LIN {X 0,Y 374.396,Z 363.23,A -85,B 0,C 180,E1 -12882.407,E2 -12882.407} C_VEL
LIN {X 0,Y 374.739,Z 351.061,A -85,B 0,C 180,E1 -12882.778,E2 -12882.778} C_VEL
LIN {X 0,Y 374.257,Z 345.258,A -85,B 0,C 180,E1 -12882.93,E2 -12882.93} C_VEL
LIN {X 0,Y 369.029,Z 326.535,A -85,B 0,C 180,E1 -12883.548,E2 -12883.548} C_VEL
LIN {X 0,Y 368.498,Z 320.718,A -85,B 0,C 180,E1 -12883.688,E2 -12883.688} C_VEL
LIN {X 0,Y 369.139,Z 272.21,A -85,B 0,C 180,E1 -12884.631,E2 -12884.631} C_VEL
LIN {X 0,Y 364.648,Z 248.183,A -85,B 0,C 180,E1 -12885.359,E2 -12885.359} C_VEL
LIN {X 0,Y 364.36,Z 246.734,A -85,B 0,C 180,E1 -12885.446,E2 -12885.446} C_VEL
LIN {X 0,Y 361.947,Z 234.402,A -85,B 0,C 180,E1 -12888.759,E2 -12888.759} C_VEL
LIN {X 0,Y 361.881,Z 234.409,A -85,B 0,C 180,E1 -12892.856,E2 -12892.856} C_VEL
LIN {X 0,Y 361.903,Z 234.406,A -85,B 0,C 180,E1 -12896.529,E2 -12896.529} C_VEL
LIN {X 0,Y 361.869,Z 234.408,A -85,B 0,C 180,E1 -12900.328,E2 -12900.328} C_VEL
LIN {X 0,Y 361.856,Z 234.409,A -85,B 0,C 180,E1 -12904.28,E2 -12904.28} C_VEL
LIN {X 0,Y 361.865,Z 234.407,A -85,B 0,C 180,E1 -12907.223,E2 -12907.223} C_VEL
LIN {X 0,Y 361.837,Z 234.415,A -85,B 0,C 180,E1 -12910.755,E2 -12910.755} C_VEL
LIN {X 0,Y 361.847,Z 234.411,A -85,B 0,C 180,E1 -12914.364,E2 -12914.364} C_VEL
LIN {X 0,Y 361.836,Z 234.409,A -85,B 0,C 180,E1 -12917.568,E2 -12917.568} C_VEL
LIN {X 0,Y 361.867,Z 234.409,A -85,B 0,C 180,E1 -12920.974,E2 -12920.974} C_VEL
LIN {X 0,Y 361.875,Z 234.411,A -85,B 0,C 180,E1 -12924.655,E2 -12924.655} C_VEL
LIN {X 0,Y 361.839,Z 234.413,A -85,B 0,C 180,E1 -12928.37,E2 -12928.37} C_VEL
LIN {X 0,Y 361.909,Z 234.403,A -85,B 0,C 180,E1 -12932.221,E2 -12932.221} C_VEL
LIN {X 0,Y 361.928,Z 234.404,A -85,B 0,C 180,E1 -12934.71,E2 -12934.71} C_VEL
LIN {X 0,Y 361.894,Z 234.406,A -85,B 0,C 180,E1 -12938.347,E2 -12938.347} C_VEL
LIN {X 0,Y 361.968,Z 234.394,A -85,B 0,C 180,E1 -12942.061,E2 -12942.061} C_VEL
LIN {X 0,Y 361.999,Z 234.391,A -85,B 0,C 180,E1 -12946.101,E2 -12946.101} C_VEL
LIN {X 0,Y 362.001,Z 234.39,A -85,B 0,C 180,E1 -12949.937,E2 -12949.937} C_VEL
LIN {X 0,Y 362.136,Z 234.373,A -85,B 0,C 180,E1 -12953.313,E2 -12953.313} C_VEL
LIN {X 0,Y 362.281,Z 234.354,A -85,B 0,C 180,E1 -12957.776,E2 -12957.776} C_VEL
LIN {X 0,Y 362.425,Z 234.337,A -85,B 0,C 180,E1 -12960,E2 -12960} C_VEL
LIN {X 0,Y 362.278,Z 234.357,A -85,B 0,C 180,E1 -12962.223,E2 -12962.223} C_VEL
LIN {X 0,Y 362.173,Z 234.373,A -85,B 0,C 180,E1 -12966.686,E2 -12966.686} C_VEL
LIN {X 0,Y 362.075,Z 234.383,A -85,B 0,C 180,E1 -12968.933,E2 -12968.933} C_VEL
LIN {X 0,Y 361.96,Z 234.398,A -85,B 0,C 180,E1 -12972.332,E2 -12972.332} C_VEL
LIN {X 0,Y 361.962,Z 234.4,A -85,B 0,C 180,E1 -12974.62,E2 -12974.62} C_VEL
LIN {X 0,Y 361.911,Z 234.402,A -85,B 0,C 180,E1 -12978.102,E2 -12978.102} C_VEL
LIN {X 0,Y 361.861,Z 234.406,A -85,B 0,C 180,E1 -12981.655,E2 -12981.655} C_VEL
LIN {X 0,Y 361.894,Z 234.403,A -85,B 0,C 180,E1 -12985.293,E2 -12985.293} C_VEL
LIN {X 0,Y 361.855,Z 234.409,A -85,B 0,C 180,E1 -12989.074,E2 -12989.074} C_VEL
LIN {X 0,Y 361.849,Z 234.41,A -85,B 0,C 180,E1 -12992.945,E2 -12992.945} C_VEL
LIN {X 0,Y 361.868,Z 234.405,A -85,B 0,C 180,E1 -12995.637,E2 -12995.637} C_VEL
LIN {X 0,Y 361.826,Z 234.413,A -85,B 0,C 180,E1 -12999.018,E2 -12999.018} C_VEL
LIN {X 0,Y 361.833,Z 234.413,A -85,B 0,C 180,E1 -13002.829,E2 -13002.829} C_VEL
LIN {X 0,Y 361.818,Z 234.413,A -85,B 0,C 180,E1 -13005.947,E2 -13005.947} C_VEL
LIN {X 0,Y 361.83,Z 234.411,A -85,B 0,C 180,E1 -13009.246,E2 -13009.246} C_VEL
LIN {X 0,Y 361.87,Z 234.409,A -85,B 0,C 180,E1 -13012.776,E2 -13012.776} C_VEL
LIN {X 0,Y 361.855,Z 234.407,A -85,B 0,C 180,E1 -13015.72,E2 -13015.72} C_VEL
LIN {X 0,Y 361.874,Z 234.409,A -85,B 0,C 180,E1 -13019.672,E2 -13019.672} C_VEL
LIN {X 0,Y 361.925,Z 234.53,A -85,B 0,C 180,E1 -13021.156,E2 -13021.156} C_VEL
LIN {X 0,Y 363.889,Z 244.234,A -85,B 0,C 180,E1 -13023.627,E2 -13023.627} C_VEL
LIN {X 0,Y 365.118,Z 252.079,A -85,B 0,C 180,E1 -13025.553,E2 -13025.553} C_VEL
LIN {X 0,Y 364.017,Z 265.513,A -85,B 0,C 180,E1 -13028.609,E2 -13028.609} C_VEL
LIN {X 0,Y 368.872,Z 299.067,A -85,B 0,C 180,E1 -13029.543,E2 -13029.543} C_VEL
LIN {X 0,Y 367.713,Z 373.609,A -85,B 0,C 180,E1 -13031.005,E2 -13031.005} C_VEL
LIN {X 0,Y 367.121,Z 386.917,A -85,B 0,C 180,E1 -13031.478,E2 -13031.478} C_VEL
LIN {X 0,Y 366.35,Z 399.141,A -85,B 0,C 180,E1 -13032.125,E2 -13032.125} C_VEL
LIN {X 0,Y 365.487,Z 410.647,A -85,B 0,C 180,E1 -13032.948,E2 -13032.948} C_VEL
LIN {X 0,Y 364.414,Z 422.442,A -85,B 0,C 180,E1 -13034.049,E2 -13034.049} C_VEL
LIN {X 0,Y 363.531,Z 432.403,A -85,B 0,C 180,E1 -13035.218,E2 -13035.218} C_VEL
LIN {X 0,Y 362.727,Z 441.68,A -85,B 0,C 180,E1 -13036.555,E2 -13036.555} C_VEL
LIN {X 0,Y 361.986,Z 449.644,A -85,B 0,C 180,E1 -13037.953,E2 -13037.953} C_VEL
LIN {X 0,Y 361.295,Z 457.417,A -85,B 0,C 180,E1 -13039.634,E2 -13039.634} C_VEL
LIN {X 0,Y 360.779,Z 464.561,A -85,B 0,C 180,E1 -13041.599,E2 -13041.599} C_VEL
LIN {X 0,Y 360.498,Z 469.31,A -85,B 0,C 180,E1 -13043.283,E2 -13043.283} C_VEL
LIN {X 0,Y 360.35,Z 472.934,A -85,B 0,C 180,E1 -13044.965,E2 -13044.965} C_VEL
LIN {X 0,Y 360.301,Z 475.537,A -85,B 0,C 180,E1 -13046.645,E2 -13046.645} C_VEL
LIN {X 0,Y 360.266,Z 476.761,A -85,B 0,C 180,E1 -13047.764,E2 -13047.764} C_VEL
LIN {X 0,Y 360.317,Z 477.556,A -85,B 0,C 180,E1 -13048.882,E2 -13048.882} C_VEL
LIN {X 0,Y 360.359,Z 477.936,A -85,B 0,C 180,E1 -13050,E2 -13050} C_VEL
LIN {X 0,Y 360.303,Z 477.928,A -85,B 0,C 180,E1 -13051.118,E2 -13051.118} C_VEL
LIN {X 0,Y 360.262,Z 477.537,A -85,B 0,C 180,E1 -13052.236,E2 -13052.236} C_VEL
LIN {X 0,Y 360.296,Z 476.738,A -85,B 0,C 180,E1 -13053.355,E2 -13053.355} C_VEL
LIN {X 0,Y 360.348,Z 475.51,A -85,B 0,C 180,E1 -13054.474,E2 -13054.474} C_VEL
LIN {X 0,Y 360.432,Z 473.128,A -85,B 0,C 180,E1 -13056.043,E2 -13056.043} C_VEL
LIN {X 0,Y 360.699,Z 469.313,A -85,B 0,C 180,E1 -13057.839,E2 -13057.839} C_VEL
LIN {X 0,Y 361.175,Z 464.617,A -85,B 0,C 180,E1 -13059.52,E2 -13059.52} C_VEL
LIN {X 0,Y 361.972,Z 457.568,A -85,B 0,C 180,E1 -13061.479,E2 -13061.479} C_VEL
LIN {X 0,Y 362.996,Z 449.946,A -85,B 0,C 180,E1 -13063.15,E2 -13063.15} C_VEL
LIN {X 0,Y 364.15,Z 440.878,A -85,B 0,C 180,E1 -13064.737,E2 -13064.737} C_VEL
LIN {X 0,Y 365.288,Z 430.537,A -85,B 0,C 180,E1 -13066.199,E2 -13066.199} C_VEL
LIN {X 0,Y 366.645,Z 419.502,A -85,B 0,C 180,E1 -13067.428,E2 -13067.428} C_VEL
LIN {X 0,Y 367.739,Z 408.708,A -85,B 0,C 180,E1 -13068.381,E2 -13068.381} C_VEL
LIN {X 0,Y 368.907,Z 396.811,A -85,B 0,C 180,E1 -13069.186,E2 -13069.186} C_VEL
LIN {X 0,Y 369.813,Z 383.937,A -85,B 0,C 180,E1 -13069.822,E2 -13069.822} C_VEL
LIN {X 0,Y 370.412,Z 370.747,A -85,B 0,C 180,E1 -13070.235,E2 -13070.235} C_VEL
LIN {X 0,Y 371.679,Z 298.745,A -85,B 0,C 180,E1 -13071.649,E2 -13071.649} C_VEL
LIN {X 0,Y 366.907,Z 272.712,A -85,B 0,C 180,E1 -13072.526,E2 -13072.526} C_VEL
LIN {X 0,Y 365.363,Z 265.186,A -85,B 0,C 180,E1 -13072.806,E2 -13072.806} C_VEL
LIN {X 0,Y 366.337,Z 255.911,A -85,B 0,C 180,E1 -13074.965,E2 -13074.965} C_VEL
LIN {X 0,Y 364.479,Z 245.888,A -85,B 0,C 180,E1 -13077.566,E2 -13077.566} C_VEL
LIN {X 0,Y 362.218,Z 235.875,A -85,B 0,C 180,E1 -13080.296,E2 -13080.296} C_VEL
LIN {X 0,Y 361.896,Z 234.407,A -85,B 0,C 180,E1 -13080.708,E2 -13080.708} C_VEL
LIN {X 0,Y 361.855,Z 234.41,A -85,B 0,C 180,E1 -13084.28,E2 -13084.28} C_VEL
LIN {X 0,Y 361.864,Z 234.411,A -85,B 0,C 180,E1 -13087.223,E2 -13087.223} C_VEL
LIN {X 0,Y 361.835,Z 234.413,A -85,B 0,C 180,E1 -13090.755,E2 -13090.755} C_VEL
LIN {X 0,Y 361.817,Z 234.414,A -85,B 0,C 180,E1 -13094.369,E2 -13094.369} C_VEL
LIN {X 0,Y 361.831,Z 234.415,A -85,B 0,C 180,E1 -13097.569,E2 -13097.569} C_VEL
LIN {X 0,Y 361.844,Z 234.413,A -85,B 0,C 180,E1 -13101.572,E2 -13101.572} C_VEL
LIN {X 0,Y 361.874,Z 234.405,A -85,B 0,C 180,E1 -13104.655,E2 -13104.655} C_VEL
LIN {X 0,Y 361.838,Z 234.41,A -85,B 0,C 180,E1 -13108.371,E2 -13108.371} C_VEL
LIN {X 0,Y 361.866,Z 234.401,A -85,B 0,C 180,E1 -13110.952,E2 -13110.952} C_VEL
LIN {X 0,Y 361.902,Z 234.396,A -85,B 0,C 180,E1 -13114.708,E2 -13114.708} C_VEL
LIN {X 0,Y 361.862,Z 234.403,A -85,B 0,C 180,E1 -13118.345,E2 -13118.345} C_VEL
LIN {X 0,Y 361.921,Z 234.398,A -85,B 0,C 180,E1 -13122.085,E2 -13122.085} C_VEL
LIN {X 0,Y 361.963,Z 234.398,A -85,B 0,C 180,E1 -13125.38,E2 -13125.38} C_VEL
LIN {X 0,Y 361.971,Z 234.388,A -85,B 0,C 180,E1 -13128.804,E2 -13128.804} C_VEL
LIN {X 0,Y 362.125,Z 234.369,A -85,B 0,C 180,E1 -13132.192,E2 -13132.192} C_VEL
LIN {X 0,Y 362.115,Z 234.373,A -85,B 0,C 180,E1 -13134.431,E2 -13134.431} C_VEL
LIN {X 0,Y 362.272,Z 234.35,A -85,B 0,C 180,E1 -13137.776,E2 -13137.776} C_VEL
LIN {X 0,Y 362.425,Z 234.338,A -85,B 0,C 180,E1 -13140,E2 -13140} C_VEL
LIN {X 0,Y 362.279,Z 234.35,A -85,B 0,C 180,E1 -13142.224,E2 -13142.224} C_VEL
LIN {X 0,Y 362.137,Z 234.373,A -85,B 0,C 180,E1 -13146.687,E2 -13146.687} C_VEL
LIN {X 0,Y 362.001,Z 234.391,A -85,B 0,C 180,E1 -13150.063,E2 -13150.063} C_VEL
LIN {X 0,Y 361.999,Z 234.388,A -85,B 0,C 180,E1 -13153.899,E2 -13153.899} C_VEL
LIN {X 0,Y 361.929,Z 234.399,A -85,B 0,C 180,E1 -13156.934,E2 -13156.934} C_VEL
LIN {X 0,Y 361.895,Z 234.402,A -85,B 0,C 180,E1 -13160.461,E2 -13160.461} C_VEL
LIN {X 0,Y 361.895,Z 234.403,A -85,B 0,C 180,E1 -13164.113,E2 -13164.113} C_VEL
LIN {X 0,Y 361.942,Z 234.391,A -85,B 0,C 180,E1 -13166.721,E2 -13166.721} C_VEL
LIN {X 0,Y 361.874,Z 234.402,A -85,B 0,C 180,E1 -13170.328,E2 -13170.328} C_VEL
LIN {X 0,Y 361.856,Z 234.408,A -85,B 0,C 180,E1 -13174.281,E2 -13174.281} C_VEL
LIN {X 0,Y 361.871,Z 234.408,A -85,B 0,C 180,E1 -13177.224,E2 -13177.224} C_VEL
LIN {X 0,Y 361.836,Z 234.412,A -85,B 0,C 180,E1 -13180.755,E2 -13180.755} C_VEL
LIN {X 0,Y 361.821,Z 234.415,A -85,B 0,C 180,E1 -13184.368,E2 -13184.368} C_VEL
LIN {X 0,Y 361.833,Z 234.412,A -85,B 0,C 180,E1 -13187.569,E2 -13187.569} C_VEL
LIN {X 0,Y 361.846,Z 234.42,A -85,B 0,C 180,E1 -13191.572,E2 -13191.572} C_VEL
LIN {X 0,Y 361.876,Z 234.412,A -85,B 0,C 180,E1 -13194.655,E2 -13194.655} C_VEL
LIN {X 0,Y 361.89,Z 234.581,A -85,B 0,C 180,E1 -13197.638,E2 -13197.638} C_VEL
LIN {X 0,Y 364.482,Z 246.196,A -85,B 0,C 180,E1 -13200.943,E2 -13200.943} C_VEL
LIN {X 0,Y 364.656,Z 247.154,A -85,B 0,C 180,E1 -13201.195,E2 -13201.195} C_VEL
LIN {X 0,Y 368.325,Z 257.097,A -85,B 0,C 180,E1 -13201.675,E2 -13201.675} C_VEL
LIN {X 0,Y 372.157,Z 273.927,A -85,B 0,C 180,E1 -13202.297,E2 -13202.297} C_VEL
LIN {X 0,Y 370.619,Z 354.332,A -85,B 0,C 180,E1 -13203.881,E2 -13203.881} C_VEL
LIN {X 0,Y 369.973,Z 367.682,A -85,B 0,C 180,E1 -13204.358,E2 -13204.358} C_VEL
LIN {X 0,Y 369.232,Z 379.987,A -85,B 0,C 180,E1 -13205.019,E2 -13205.019} C_VEL
LIN {X 0,Y 368.134,Z 392.32,A -85,B 0,C 180,E1 -13205.916,E2 -13205.916} C_VEL
LIN {X 0,Y 367.068,Z 403.069,A -85,B 0,C 180,E1 -13206.937,E2 -13206.937} C_VEL
LIN {X 0,Y 365.742,Z 413.323,A -85,B 0,C 180,E1 -13208.142,E2 -13208.142} C_VEL
LIN {X 0,Y 364.786,Z 422.027,A -85,B 0,C 180,E1 -13209.414,E2 -13209.414} C_VEL
LIN {X 0,Y 363.735,Z 430.01,A -85,B 0,C 180,E1 -13210.824,E2 -13210.824} C_VEL
LIN {X 0,Y 362.722,Z 437.778,A -85,B 0,C 180,E1 -13212.523,E2 -13212.523} C_VEL
LIN {X 0,Y 361.904,Z 443.979,A -85,B 0,C 180,E1 -13214.224,E2 -13214.224} C_VEL
LIN {X 0,Y 361.308,Z 448.882,A -85,B 0,C 180,E1 -13215.928,E2 -13215.928} C_VEL
LIN {X 0,Y 360.865,Z 452.641,A -85,B 0,C 180,E1 -13217.63,E2 -13217.63} C_VEL
LIN {X 0,Y 360.603,Z 454.574,A -85,B 0,C 180,E1 -13218.761,E2 -13218.761} C_VEL
LIN {X 0,Y 360.406,Z 456.08,A -85,B 0,C 180,E1 -13219.892,E2 -13219.892} C_VEL
LIN {X 0,Y 360.346,Z 457.127,A -85,B 0,C 180,E1 -13221.024,E2 -13221.024} C_VEL
LIN {X 0,Y 360.356,Z 458.051,A -85,B 0,C 180,E1 -13223.28,E2 -13223.28} C_VEL
LIN {X 0,Y 360.339,Z 457.93,A -85,B 0,C 180,E1 -13224.404,E2 -13224.404} C_VEL
LIN {X 0,Y 360.337,Z 457.379,A -85,B 0,C 180,E1 -13225.525,E2 -13225.525} C_VEL
LIN {X 0,Y 360.368,Z 455.116,A -85,B 0,C 180,E1 -13227.765,E2 -13227.765} C_VEL
LIN {X 0,Y 360.561,Z 452.313,A -85,B 0,C 180,E1 -13229.442,E2 -13229.442} C_VEL
LIN {X 0,Y 360.77,Z 448.504,A -85,B 0,C 180,E1 -13231.116,E2 -13231.116} C_VEL
LIN {X 0,Y 361.196,Z 443.574,A -85,B 0,C 180,E1 -13232.788,E2 -13232.788} C_VEL
LIN {X 0,Y 361.732,Z 437.388,A -85,B 0,C 180,E1 -13234.457,E2 -13234.457} C_VEL
LIN {X 0,Y 362.497,Z 429.658,A -85,B 0,C 180,E1 -13236.121,E2 -13236.121} C_VEL
LIN {X 0,Y 363.56,Z 419.993,A -85,B 0,C 180,E1 -13237.777,E2 -13237.777} C_VEL
LIN {X 0,Y 364.5,Z 410.002,A -85,B 0,C 180,E1 -13239.153,E2 -13239.153} C_VEL
LIN {X 0,Y 365.488,Z 398.682,A -85,B 0,C 180,E1 -13240.386,E2 -13240.386} C_VEL
LIN {X 0,Y 366.334,Z 387.589,A -85,B 0,C 180,E1 -13241.341,E2 -13241.341} C_VEL
LIN {X 0,Y 367.092,Z 375.196,A -85,B 0,C 180,E1 -13242.157,E2 -13242.157} C_VEL
LIN {X 0,Y 367.633,Z 362.16,A -85,B 0,C 180,E1 -13242.762,E2 -13242.762} C_VEL
LIN {X 0,Y 367.993,Z 349.854,A -85,B 0,C 180,E1 -13243.124,E2 -13243.124} C_VEL
LIN {X 0,Y 368.498,Z 320.718,A -85,B 0,C 180,E1 -13243.688,E2 -13243.688} C_VEL
LIN {X 0,Y 367.969,Z 314.906,A -85,B 0,C 180,E1 -13243.831,E2 -13243.831} C_VEL
LIN {X 0,Y 362.777,Z 296.203,A -85,B 0,C 180,E1 -13244.477,E2 -13244.477} C_VEL
LIN {X 0,Y 362.288,Z 290.391,A -85,B 0,C 180,E1 -13244.621,E2 -13244.621} C_VEL
LIN {X 0,Y 362.466,Z 273.403,A -85,B 0,C 180,E1 -13244.961,E2 -13244.961} C_VEL
LIN {X 0,Y 358.093,Z 249.854,A -85,B 0,C 180,E1 -13245.691,E2 -13245.691} C_VEL
LIN {X 0,Y 357.227,Z 246.955,A -85,B 0,C 180,E1 -13245.837,E2 -13245.837} C_VEL
LIN {X 0,Y 354.899,Z 235.278,A -85,B 0,C 180,E1 -13249.071,E2 -13249.071} C_VEL
LIN {X 0,Y 354.818,Z 235.285,A -85,B 0,C 180,E1 -13252.107,E2 -13252.107} C_VEL
LIN {X 0,Y 354.866,Z 235.278,A -85,B 0,C 180,E1 -13255.83,E2 -13255.83} C_VEL
LIN {X 0,Y 354.809,Z 235.285,A -85,B 0,C 180,E1 -13259.683,E2 -13259.683} C_VEL
LIN {X 0,Y 354.816,Z 235.284,A -85,B 0,C 180,E1 -13263.684,E2 -13263.684} C_VEL
LIN {X 0,Y 354.8,Z 235.29,A -85,B 0,C 180,E1 -13266.459,E2 -13266.459} C_VEL
LIN {X 0,Y 354.826,Z 235.283,A -85,B 0,C 180,E1 -13269.423,E2 -13269.423} C_VEL
LIN {X 0,Y 354.79,Z 235.291,A -85,B 0,C 180,E1 -13272.867,E2 -13272.867} C_VEL
LIN {X 0,Y 354.769,Z 235.291,A -85,B 0,C 180,E1 -13276.104,E2 -13276.104} C_VEL
LIN {X 0,Y 354.786,Z 235.289,A -85,B 0,C 180,E1 -13279.178,E2 -13279.178} C_VEL
LIN {X 0,Y 354.807,Z 235.289,A -85,B 0,C 180,E1 -13282.402,E2 -13282.402} C_VEL
LIN {X 0,Y 354.813,Z 235.288,A -85,B 0,C 180,E1 -13284.941,E2 -13284.941} C_VEL
LIN {X 0,Y 354.794,Z 235.29,A -85,B 0,C 180,E1 -13288.405,E2 -13288.405} C_VEL
LIN {X 0,Y 354.847,Z 235.28,A -85,B 0,C 180,E1 -13291.618,E2 -13291.618} C_VEL
LIN {X 0,Y 354.899,Z 235.275,A -85,B 0,C 180,E1 -13294.172,E2 -13294.172} C_VEL
LIN {X 0,Y 354.837,Z 235.282,A -85,B 0,C 180,E1 -13297.894,E2 -13297.894} C_VEL
LIN {X 0,Y 354.923,Z 235.271,A -85,B 0,C 180,E1 -13301.891,E2 -13301.891} C_VEL
LIN {X 0,Y 354.943,Z 235.269,A -85,B 0,C 180,E1 -13305.981,E2 -13305.981} C_VEL
LIN {X 0,Y 354.957,Z 235.266,A -85,B 0,C 180,E1 -13309.735,E2 -13309.735} C_VEL
LIN {X 0,Y 355.099,Z 235.25,A -85,B 0,C 180,E1 -13313.18,E2 -13313.18} C_VEL
LIN {X 0,Y 355.244,Z 235.231,A -85,B 0,C 180,E1 -13317.732,E2 -13317.732} C_VEL
LIN {X 0,Y 355.374,Z 235.215,A -85,B 0,C 180,E1 -13320,E2 -13320} C_VEL
LIN {X 0,Y 355.241,Z 235.234,A -85,B 0,C 180,E1 -13322.268,E2 -13322.268} C_VEL
LIN {X 0,Y 355.139,Z 235.248,A -85,B 0,C 180,E1 -13326.819,E2 -13326.819} C_VEL
LIN {X 0,Y 355.016,Z 235.261,A -85,B 0,C 180,E1 -13329.112,E2 -13329.112} C_VEL
LIN {X 0,Y 354.922,Z 235.277,A -85,B 0,C 180,E1 -13332.581,E2 -13332.581} C_VEL
LIN {X 0,Y 354.888,Z 235.277,A -85,B 0,C 180,E1 -13336.096,E2 -13336.096} C_VEL
LIN {X 0,Y 354.844,Z 235.28,A -85,B 0,C 180,E1 -13339.676,E2 -13339.676} C_VEL
LIN {X 0,Y 354.825,Z 235.283,A -85,B 0,C 180,E1 -13343.337,E2 -13343.337} C_VEL
LIN {X 0,Y 354.814,Z 235.287,A -85,B 0,C 180,E1 -13346.958,E2 -13346.958} C_VEL
LIN {X 0,Y 354.799,Z 235.286,A -85,B 0,C 180,E1 -13349.684,E2 -13349.684} C_VEL
LIN {X 0,Y 354.787,Z 235.291,A -85,B 0,C 180,E1 -13352.333,E2 -13352.333} C_VEL
LIN {X 0,Y 354.822,Z 235.283,A -85,B 0,C 180,E1 -13355.699,E2 -13355.699} C_VEL
LIN {X 0,Y 354.768,Z 235.29,A -85,B 0,C 180,E1 -13359.413,E2 -13359.413} C_VEL
LIN {X 0,Y 354.786,Z 235.291,A -85,B 0,C 180,E1 -13362.867,E2 -13362.867} C_VEL
LIN {X 0,Y 354.767,Z 235.292,A -85,B 0,C 180,E1 -13366.104,E2 -13366.104} C_VEL
LIN {X 0,Y 354.782,Z 235.289,A -85,B 0,C 180,E1 -13369.178,E2 -13369.178} C_VEL
LIN {X 0,Y 354.811,Z 235.29,A -85,B 0,C 180,E1 -13372.402,E2 -13372.402} C_VEL
LIN {X 0,Y 354.812,Z 235.287,A -85,B 0,C 180,E1 -13374.941,E2 -13374.941} C_VEL
LIN {X 0,Y 354.794,Z 235.292,A -85,B 0,C 180,E1 -13378.405,E2 -13378.405} C_VEL
LIN {X 0,Y 354.879,Z 235.478,A -85,B 0,C 180,E1 -13380.875,E2 -13380.875} C_VEL
LIN {X 0,Y 356.852,Z 245.099,A -85,B 0,C 180,E1 -13383.382,E2 -13383.382} C_VEL
LIN {X 0,Y 358.18,Z 253.083,A -85,B 0,C 180,E1 -13385.389,E2 -13385.389} C_VEL
LIN {X 0,Y 357.143,Z 265.309,A -85,B 0,C 180,E1 -13388.226,E2 -13388.226} C_VEL
LIN {X 0,Y 362.12,Z 299.306,A -85,B 0,C 180,E1 -13389.2,E2 -13389.2} C_VEL
LIN {X 0,Y 360.906,Z 374.206,A -85,B 0,C 180,E1 -13390.705,E2 -13390.705} C_VEL
LIN {X 0,Y 360.227,Z 388.055,A -85,B 0,C 180,E1 -13391.221,E2 -13391.221} C_VEL
LIN {X 0,Y 359.396,Z 400.464,A -85,B 0,C 180,E1 -13391.915,E2 -13391.915} C_VEL
LIN {X 0,Y 358.382,Z 413.153,A -85,B 0,C 180,E1 -13392.893,E2 -13392.893} C_VEL
LIN {X 0,Y 357.306,Z 424.442,A -85,B 0,C 180,E1 -13394.016,E2 -13394.016} C_VEL
LIN {X 0,Y 356.44,Z 434.602,A -85,B 0,C 180,E1 -13395.294,E2 -13395.294} C_VEL
LIN {X 0,Y 355.514,Z 444.586,A -85,B 0,C 180,E1 -13396.86,E2 -13396.86} C_VEL
LIN {X 0,Y 354.538,Z 453.355,A -85,B 0,C 180,E1 -13398.567,E2 -13398.567} C_VEL
LIN {X 0,Y 353.992,Z 460.351,A -85,B 0,C 180,E1 -13400.285,E2 -13400.285} C_VEL
LIN {X 0,Y 353.605,Z 465.948,A -85,B 0,C 180,E1 -13402.003,E2 -13402.003} C_VEL
LIN {X 0,Y 353.33,Z 470.97,A -85,B 0,C 180,E1 -13404.009,E2 -13404.009} C_VEL
LIN {X 0,Y 353.279,Z 473.644,A -85,B 0,C 180,E1 -13405.436,E2 -13405.436} C_VEL
LIN {X 0,Y 353.223,Z 475.285,A -85,B 0,C 180,E1 -13406.578,E2 -13406.578} C_VEL
LIN {X 0,Y 353.174,Z 476.522,A -85,B 0,C 180,E1 -13407.719,E2 -13407.719} C_VEL
LIN {X 0,Y 353.217,Z 477.341,A -85,B 0,C 180,E1 -13408.86,E2 -13408.86} C_VEL
LIN {X 0,Y 353.262,Z 477.733,A -85,B 0,C 180,E1 -13410,E2 -13410} C_VEL
LIN {X 0,Y 353.17,Z 477.359,A -85,B 0,C 180,E1 -13412.281,E2 -13412.281} C_VEL
LIN {X 0,Y 353.217,Z 476.583,A -85,B 0,C 180,E1 -13413.422,E2 -13413.422} C_VEL
LIN {X 0,Y 353.263,Z 475.369,A -85,B 0,C 180,E1 -13414.564,E2 -13414.564} C_VEL
LIN {X 0,Y 353.323,Z 473.326,A -85,B 0,C 180,E1 -13415.979,E2 -13415.979} C_VEL
LIN {X 0,Y 353.64,Z 469.225,A -85,B 0,C 180,E1 -13417.997,E2 -13417.997} C_VEL
LIN {X 0,Y 354.134,Z 464.56,A -85,B 0,C 180,E1 -13419.712,E2 -13419.712} C_VEL
LIN {X 0,Y 354.975,Z 457.545,A -85,B 0,C 180,E1 -13421.709,E2 -13421.709} C_VEL
LIN {X 0,Y 356.07,Z 449.967,A -85,B 0,C 180,E1 -13423.41,E2 -13423.41} C_VEL
LIN {X 0,Y 357.249,Z 441.113,A -85,B 0,C 180,E1 -13425.003,E2 -13425.003} C_VEL
LIN {X 0,Y 358.463,Z 430.675,A -85,B 0,C 180,E1 -13426.516,E2 -13426.516} C_VEL
LIN {X 0,Y 359.875,Z 419.752,A -85,B 0,C 180,E1 -13427.767,E2 -13427.767} C_VEL
LIN {X 0,Y 361.018,Z 409.066,A -85,B 0,C 180,E1 -13428.736,E2 -13428.736} C_VEL
LIN {X 0,Y 362.295,Z 396.202,A -85,B 0,C 180,E1 -13429.623,E2 -13429.623} C_VEL
LIN {X 0,Y 363.28,Z 383.084,A -85,B 0,C 180,E1 -13430.268,E2 -13430.268} C_VEL
LIN {X 0,Y 363.861,Z 369.479,A -85,B 0,C 180,E1 -13430.689,E2 -13430.689} C_VEL
LIN {X 0,Y 365.199,Z 299.874,A -85,B 0,C 180,E1 -13432.073,E2 -13432.073} C_VEL
LIN {X 0,Y 360.474,Z 273.805,A -85,B 0,C 180,E1 -13432.971,E2 -13432.971} C_VEL
LIN {X 0,Y 358.646,Z 264.966,A -85,B 0,C 180,E1 -13433.313,E2 -13433.313} C_VEL
LIN {X 0,Y 359.444,Z 257.174,A -85,B 0,C 180,E1 -13435.168,E2 -13435.168} C_VEL
LIN {X 0,Y 357.296,Z 245.902,A -85,B 0,C 180,E1 -13438.169,E2 -13438.169} C_VEL
LIN {X 0,Y 354.811,Z 235.289,A -85,B 0,C 180,E1 -13441.217,E2 -13441.217} C_VEL
LIN {X 0,Y 354.813,Z 235.286,A -85,B 0,C 180,E1 -13445.059,E2 -13445.059} C_VEL
LIN {X 0,Y 354.806,Z 235.29,A -85,B 0,C 180,E1 -13447.883,E2 -13447.883} C_VEL
LIN {X 0,Y 354.787,Z 235.292,A -85,B 0,C 180,E1 -13451.171,E2 -13451.171} C_VEL
LIN {X 0,Y 354.764,Z 235.293,A -85,B 0,C 180,E1 -13454.506,E2 -13454.506} C_VEL
LIN {X 0,Y 354.789,Z 235.293,A -85,B 0,C 180,E1 -13457.662,E2 -13457.662} C_VEL
LIN {X 0,Y 354.785,Z 235.289,A -85,B 0,C 180,E1 -13460.662,E2 -13460.662} C_VEL
LIN {X 0,Y 354.822,Z 235.284,A -85,B 0,C 180,E1 -13464.301,E2 -13464.301} C_VEL
LIN {X 0,Y 354.787,Z 235.29,A -85,B 0,C 180,E1 -13467.667,E2 -13467.667} C_VEL
LIN {X 0,Y 354.811,Z 235.287,A -85,B 0,C 180,E1 -13471.615,E2 -13471.615} C_VEL
LIN {X 0,Y 354.854,Z 235.279,A -85,B 0,C 180,E1 -13475.423,E2 -13475.423} C_VEL
LIN {X 0,Y 354.827,Z 235.28,A -85,B 0,C 180,E1 -13479.113,E2 -13479.113} C_VEL
LIN {X 0,Y 354.881,Z 235.275,A -85,B 0,C 180,E1 -13482.719,E2 -13482.719} C_VEL
LIN {X 0,Y 354.952,Z 235.267,A -85,B 0,C 180,E1 -13486.255,E2 -13486.255} C_VEL
LIN {X 0,Y 354.978,Z 235.267,A -85,B 0,C 180,E1 -13489.736,E2 -13489.736} C_VEL
LIN {X 0,Y 355.128,Z 235.241,A -85,B 0,C 180,E1 -13493.181,E2 -13493.181} C_VEL
LIN {X 0,Y 355.234,Z 235.226,A -85,B 0,C 180,E1 -13497.732,E2 -13497.732} C_VEL
LIN {X 0,Y 355.374,Z 235.216,A -85,B 0,C 180,E1 -13500,E2 -13500} C_VEL
LIN {X 0,Y 355.242,Z 235.227,A -85,B 0,C 180,E1 -13502.268,E2 -13502.268} C_VEL
LIN {X 0,Y 355.101,Z 235.25,A -85,B 0,C 180,E1 -13506.82,E2 -13506.82} C_VEL
LIN {X 0,Y 354.957,Z 235.268,A -85,B 0,C 180,E1 -13510.265,E2 -13510.265} C_VEL
LIN {X 0,Y 354.944,Z 235.267,A -85,B 0,C 180,E1 -13514.019,E2 -13514.019} C_VEL
LIN {X 0,Y 354.891,Z 235.269,A -85,B 0,C 180,E1 -13518.092,E2 -13518.092} C_VEL
LIN {X 0,Y 354.836,Z 235.275,A -85,B 0,C 180,E1 -13522.106,E2 -13522.106} C_VEL
LIN {X 0,Y 354.9,Z 235.27,A -85,B 0,C 180,E1 -13525.828,E2 -13525.828} C_VEL
LIN {X 0,Y 354.819,Z 235.283,A -85,B 0,C 180,E1 -13529.682,E2 -13529.682} C_VEL
LIN {X 0,Y 354.808,Z 235.287,A -85,B 0,C 180,E1 -13533.702,E2 -13533.702} C_VEL
LIN {X 0,Y 354.801,Z 235.284,A -85,B 0,C 180,E1 -13536.459,E2 -13536.459} C_VEL
LIN {X 0,Y 354.826,Z 235.286,A -85,B 0,C 180,E1 -13539.424,E2 -13539.424} C_VEL
LIN {X 0,Y 354.789,Z 235.291,A -85,B 0,C 180,E1 -13542.867,E2 -13542.867} C_VEL
LIN {X 0,Y 354.782,Z 235.286,A -85,B 0,C 180,E1 -13546.106,E2 -13546.106} C_VEL
LIN {X 0,Y 354.768,Z 235.298,A -85,B 0,C 180,E1 -13549.176,E2 -13549.176} C_VEL
LIN {X 0,Y 354.802,Z 235.293,A -85,B 0,C 180,E1 -13552.404,E2 -13552.404} C_VEL
LIN {X 0,Y 354.814,Z 235.291,A -85,B 0,C 180,E1 -13554.941,E2 -13554.941} C_VEL
LIN {X 0,Y 354.84,Z 235.343,A -85,B 0,C 180,E1 -13557.167,E2 -13557.167} C_VEL
LIN {X 0,Y 357.485,Z 247.252,A -85,B 0,C 180,E1 -13560.635,E2 -13560.635} C_VEL
LIN {X 0,Y 362.074,Z 259.165,A -85,B 0,C 180,E1 -13561.26,E2 -13561.26} C_VEL
LIN {X 0,Y 365.7,Z 275.209,A -85,B 0,C 180,E1 -13561.869,E2 -13561.869} C_VEL
LIN {X 0,Y 364.068,Z 354.88,A -85,B 0,C 180,E1 -13563.467,E2 -13563.467} C_VEL
LIN {X 0,Y 363.376,Z 368.586,A -85,B 0,C 180,E1 -13563.973,E2 -13563.973} C_VEL
LIN {X 0,Y 362.554,Z 381.262,A -85,B 0,C 180,E1 -13564.68,E2 -13564.68} C_VEL
LIN {X 0,Y 361.405,Z 393.279,A -85,B 0,C 180,E1 -13565.592,E2 -13565.592} C_VEL
LIN {X 0,Y 360.31,Z 403.71,A -85,B 0,C 180,E1 -13566.61,E2 -13566.61} C_VEL
LIN {X 0,Y 358.918,Z 414.032,A -85,B 0,C 180,E1 -13567.856,E2 -13567.856} C_VEL
LIN {X 0,Y 357.815,Z 423.515,A -85,B 0,C 180,E1 -13569.296,E2 -13569.296} C_VEL
LIN {X 0,Y 356.614,Z 432.253,A -85,B 0,C 180,E1 -13570.944,E2 -13570.944} C_VEL
LIN {X 0,Y 355.541,Z 439.927,A -85,B 0,C 180,E1 -13572.752,E2 -13572.752} C_VEL
LIN {X 0,Y 354.726,Z 445.748,A -85,B 0,C 180,E1 -13574.486,E2 -13574.486} C_VEL
LIN {X 0,Y 354.04,Z 451.077,A -85,B 0,C 180,E1 -13576.581,E2 -13576.581} C_VEL
LIN {X 0,Y 353.568,Z 454.653,A -85,B 0,C 180,E1 -13578.535,E2 -13578.535} C_VEL
LIN {X 0,Y 353.339,Z 456.19,A -85,B 0,C 180,E1 -13579.688,E2 -13579.688} C_VEL
LIN {X 0,Y 353.254,Z 457.272,A -85,B 0,C 180,E1 -13580.842,E2 -13580.842} C_VEL
LIN {X 0,Y 353.269,Z 458.238,A -85,B 0,C 180,E1 -13583.144,E2 -13583.144} C_VEL
LIN {X 0,Y 353.263,Z 458.147,A -85,B 0,C 180,E1 -13584.291,E2 -13584.291} C_VEL
LIN {X 0,Y 353.25,Z 457.629,A -85,B 0,C 180,E1 -13585.435,E2 -13585.435} C_VEL
LIN {X 0,Y 353.268,Z 455.409,A -85,B 0,C 180,E1 -13587.72,E2 -13587.72} C_VEL
LIN {X 0,Y 353.486,Z 452.649,A -85,B 0,C 180,E1 -13589.43,E2 -13589.43} C_VEL
LIN {X 0,Y 353.697,Z 448.887,A -85,B 0,C 180,E1 -13591.139,E2 -13591.139} C_VEL
LIN {X 0,Y 354.119,Z 444.009,A -85,B 0,C 180,E1 -13592.844,E2 -13592.844} C_VEL
LIN {X 0,Y 354.683,Z 437.877,A -85,B 0,C 180,E1 -13594.546,E2 -13594.546} C_VEL
LIN {X 0,Y 355.47,Z 430.243,A -85,B 0,C 180,E1 -13596.243,E2 -13596.243} C_VEL
LIN {X 0,Y 356.556,Z 420.655,A -85,B 0,C 180,E1 -13597.931,E2 -13597.931} C_VEL
LIN {X 0,Y 357.547,Z 410.776,A -85,B 0,C 180,E1 -13599.332,E2 -13599.332} C_VEL
LIN {X 0,Y 358.558,Z 399.62,A -85,B 0,C 180,E1 -13600.589,E2 -13600.589} C_VEL
LIN {X 0,Y 359.444,Z 388.703,A -85,B 0,C 180,E1 -13601.561,E2 -13601.561} C_VEL
LIN {X 0,Y 360.244,Z 376.624,A -85,B 0,C 180,E1 -13602.392,E2 -13602.392} C_VEL
LIN {X 0,Y 360.782,Z 364.261,A -85,B 0,C 180,E1 -13603.009,E2 -13603.009} C_VEL
LIN {X 0,Y 361.174,Z 351.739,A -85,B 0,C 180,E1 -13603.411,E2 -13603.411} C_VEL
LIN {X 0,Y 362.288,Z 290.391,A -85,B 0,C 180,E1 -13604.621,E2 -13604.621} C_VEL
LIN {X 0,Y 362.058,Z 286.498,A -85,B 0,C 180,E1 -13604.714,E2 -13604.714} C_VEL
LIN {X 0,Y 360.714,Z 280.835,A -85,B 0,C 180,E1 -13604.902,E2 -13604.902} C_VEL
LIN {X 0,Y 354.331,Z 264.445,A -85,B 0,C 180,E1 -13605.599,E2 -13605.599} C_VEL
LIN {X 0,Y 353.377,Z 260.618,A -85,B 0,C 180,E1 -13605.735,E2 -13605.735} C_VEL
LIN {X 0,Y 350.987,Z 249.944,A -85,B 0,C 180,E1 -13606.101,E2 -13606.101} C_VEL
LIN {X 0,Y 350.053,Z 247.271,A -85,B 0,C 180,E1 -13606.223,E2 -13606.223} C_VEL
LIN {X 0,Y 347.841,Z 236.157,A -85,B 0,C 180,E1 -13609.359,E2 -13609.359} C_VEL
LIN {X 0,Y 347.764,Z 236.168,A -85,B 0,C 180,E1 -13612.58,E2 -13612.58} C_VEL
LIN {X 0,Y 347.795,Z 236.161,A -85,B 0,C 180,E1 -13615.11,E2 -13615.11} C_VEL
LIN {X 0,Y 347.759,Z 236.166,A -85,B 0,C 180,E1 -13619.014,E2 -13619.014} C_VEL
LIN {X 0,Y 347.735,Z 236.169,A -85,B 0,C 180,E1 -13623.072,E2 -13623.072} C_VEL
LIN {X 0,Y 347.772,Z 236.162,A -85,B 0,C 180,E1 -13626.065,E2 -13626.065} C_VEL
LIN {X 0,Y 347.754,Z 236.169,A -85,B 0,C 180,E1 -13628.792,E2 -13628.792} C_VEL
LIN {X 0,Y 347.752,Z 236.164,A -85,B 0,C 180,E1 -13631.83,E2 -13631.83} C_VEL
LIN {X 0,Y 347.767,Z 236.165,A -85,B 0,C 180,E1 -13635.017,E2 -13635.017} C_VEL
LIN {X 0,Y 347.75,Z 236.168,A -85,B 0,C 180,E1 -13638.397,E2 -13638.397} C_VEL
LIN {X 0,Y 347.774,Z 236.162,A -85,B 0,C 180,E1 -13642.011,E2 -13642.011} C_VEL
LIN {X 0,Y 347.745,Z 236.165,A -85,B 0,C 180,E1 -13645.536,E2 -13645.536} C_VEL
LIN {X 0,Y 347.746,Z 236.166,A -85,B 0,C 180,E1 -13648.3,E2 -13648.3} C_VEL
LIN {X 0,Y 347.779,Z 236.163,A -85,B 0,C 180,E1 -13650.987,E2 -13650.987} C_VEL
LIN {X 0,Y 347.831,Z 236.154,A -85,B 0,C 180,E1 -13653.607,E2 -13653.607} C_VEL
LIN {X 0,Y 347.79,Z 236.16,A -85,B 0,C 180,E1 -13656.162,E2 -13656.162} C_VEL
LIN {X 0,Y 347.813,Z 236.156,A -85,B 0,C 180,E1 -13659.909,E2 -13659.909} C_VEL
LIN {X 0,Y 347.867,Z 236.153,A -85,B 0,C 180,E1 -13662.359,E2 -13662.359} C_VEL
LIN {X 0,Y 347.898,Z 236.146,A -85,B 0,C 180,E1 -13665.971,E2 -13665.971} C_VEL
LIN {X 0,Y 347.897,Z 236.145,A -85,B 0,C 180,E1 -13669.524,E2 -13669.524} C_VEL
LIN {X 0,Y 348.064,Z 236.127,A -85,B 0,C 180,E1 -13673.041,E2 -13673.041} C_VEL
LIN {X 0,Y 348.206,Z 236.107,A -85,B 0,C 180,E1 -13677.686,E2 -13677.686} C_VEL
LIN {X 0,Y 348.324,Z 236.094,A -85,B 0,C 180,E1 -13680,E2 -13680} C_VEL
LIN {X 0,Y 348.203,Z 236.111,A -85,B 0,C 180,E1 -13682.313,E2 -13682.313} C_VEL
LIN {X 0,Y 348.107,Z 236.122,A -85,B 0,C 180,E1 -13686.958,E2 -13686.958} C_VEL
LIN {X 0,Y 347.968,Z 236.137,A -85,B 0,C 180,E1 -13689.298,E2 -13689.298} C_VEL
LIN {X 0,Y 347.89,Z 236.15,A -85,B 0,C 180,E1 -13692.839,E2 -13692.839} C_VEL
LIN {X 0,Y 347.833,Z 236.159,A -85,B 0,C 180,E1 -13696.432,E2 -13696.432} C_VEL
LIN {X 0,Y 347.8,Z 236.159,A -85,B 0,C 180,E1 -13700.091,E2 -13700.091} C_VEL
LIN {X 0,Y 347.774,Z 236.161,A -85,B 0,C 180,E1 -13703.839,E2 -13703.839} C_VEL
LIN {X 0,Y 347.741,Z 236.165,A -85,B 0,C 180,E1 -13707.7,E2 -13707.7} C_VEL
LIN {X 0,Y 347.741,Z 236.169,A -85,B 0,C 180,E1 -13710.349,E2 -13710.349} C_VEL
LIN {X 0,Y 347.748,Z 236.166,A -85,B 0,C 180,E1 -13714.044,E2 -13714.044} C_VEL
LIN {X 0,Y 347.757,Z 236.164,A -85,B 0,C 180,E1 -13717.321,E2 -13717.321} C_VEL
LIN {X 0,Y 347.742,Z 236.165,A -85,B 0,C 180,E1 -13721.601,E2 -13721.601} C_VEL
LIN {X 0,Y 347.706,Z 236.171,A -85,B 0,C 180,E1 -13725.027,E2 -13725.027} C_VEL
LIN {X 0,Y 347.747,Z 236.169,A -85,B 0,C 180,E1 -13728.398,E2 -13728.398} C_VEL
LIN {X 0,Y 347.776,Z 236.162,A -85,B 0,C 180,E1 -13732.011,E2 -13732.011} C_VEL
LIN {X 0,Y 347.745,Z 236.165,A -85,B 0,C 180,E1 -13735.536,E2 -13735.536} C_VEL
LIN {X 0,Y 347.746,Z 236.169,A -85,B 0,C 180,E1 -13738.301,E2 -13738.301} C_VEL
LIN {X 0,Y 347.82,Z 236.261,A -85,B 0,C 180,E1 -13740.541,E2 -13740.541} C_VEL
LIN {X 0,Y 349.841,Z 245.961,A -85,B 0,C 180,E1 -13743.128,E2 -13743.128} C_VEL
LIN {X 0,Y 351.188,Z 253.818,A -85,B 0,C 180,E1 -13745.149,E2 -13745.149} C_VEL
LIN {X 0,Y 350.32,Z 264.095,A -85,B 0,C 180,E1 -13747.594,E2 -13747.594} C_VEL
LIN {X 0,Y 350.23,Z 265.054,A -85,B 0,C 180,E1 -13747.82,E2 -13747.82} C_VEL
LIN {X 0,Y 355.391,Z 300.222,A -85,B 0,C 180,E1 -13748.859,E2 -13748.859} C_VEL
LIN {X 0,Y 354.152,Z 373.702,A -85,B 0,C 180,E1 -13750.36,E2 -13750.36} C_VEL
LIN {X 0,Y 353.495,Z 386.888,A -85,B 0,C 180,E1 -13750.85,E2 -13750.85} C_VEL
LIN {X 0,Y 352.623,Z 399.586,A -85,B 0,C 180,E1 -13751.555,E2 -13751.555} C_VEL
LIN {X 0,Y 351.714,Z 410.861,A -85,B 0,C 180,E1 -13752.408,E2 -13752.408} C_VEL
LIN {X 0,Y 350.597,Z 422.535,A -85,B 0,C 180,E1 -13753.552,E2 -13753.552} C_VEL
LIN {X 0,Y 349.545,Z 433.038,A -85,B 0,C 180,E1 -13754.848,E2 -13754.848} C_VEL
LIN {X 0,Y 348.687,Z 442.487,A -85,B 0,C 180,E1 -13756.301,E2 -13756.301} C_VEL
LIN {X 0,Y 347.704,Z 451.59,A -85,B 0,C 180,E1 -13758.043,E2 -13758.043} C_VEL
LIN {X 0,Y 347.045,Z 458.925,A -85,B 0,C 180,E1 -13759.794,E2 -13759.794} C_VEL
LIN {X 0,Y 346.666,Z 463.884,A -85,B 0,C 180,E1 -13761.254,E2 -13761.254} C_VEL
LIN {X 0,Y 346.341,Z 468.694,A -85,B 0,C 180,E1 -13763.007,E2 -13763.007} C_VEL
LIN {X 0,Y 346.201,Z 471.879,A -85,B 0,C 180,E1 -13764.488,E2 -13764.488} C_VEL
LIN {X 0,Y 346.147,Z 475.033,A -85,B 0,C 180,E1 -13766.508,E2 -13766.508} C_VEL
LIN {X 0,Y 346.086,Z 476.281,A -85,B 0,C 180,E1 -13767.672,E2 -13767.672} C_VEL
LIN {X 0,Y 346.117,Z 477.124,A -85,B 0,C 180,E1 -13768.837,E2 -13768.837} C_VEL
LIN {X 0,Y 346.165,Z 477.531,A -85,B 0,C 180,E1 -13770,E2 -13770} C_VEL
LIN {X 0,Y 346.082,Z 477.181,A -85,B 0,C 180,E1 -13772.328,E2 -13772.328} C_VEL
LIN {X 0,Y 346.141,Z 476.425,A -85,B 0,C 180,E1 -13773.492,E2 -13773.492} C_VEL
LIN {X 0,Y 346.163,Z 475.228,A -85,B 0,C 180,E1 -13774.658,E2 -13774.658} C_VEL
LIN {X 0,Y 346.242,Z 473.423,A -85,B 0,C 180,E1 -13775.956,E2 -13775.956} C_VEL
LIN {X 0,Y 346.584,Z 469.14,A -85,B 0,C 180,E1 -13778.16,E2 -13778.16} C_VEL
LIN {X 0,Y 347.107,Z 464.504,A -85,B 0,C 180,E1 -13779.91,E2 -13779.91} C_VEL
LIN {X 0,Y 348.001,Z 457.523,A -85,B 0,C 180,E1 -13781.947,E2 -13781.947} C_VEL
LIN {X 0,Y 349.158,Z 449.984,A -85,B 0,C 180,E1 -13783.681,E2 -13783.681} C_VEL
LIN {X 0,Y 350.222,Z 442.298,A -85,B 0,C 180,E1 -13785.122,E2 -13785.122} C_VEL
LIN {X 0,Y 351.526,Z 431.885,A -85,B 0,C 180,E1 -13786.702,E2 -13786.702} C_VEL
LIN {X 0,Y 352.998,Z 421.294,A -85,B 0,C 180,E1 -13787.975,E2 -13787.975} C_VEL
LIN {X 0,Y 354.323,Z 409.432,A -85,B 0,C 180,E1 -13789.104,E2 -13789.104} C_VEL
LIN {X 0,Y 355.654,Z 396.723,A -85,B 0,C 180,E1 -13790.005,E2 -13790.005} C_VEL
LIN {X 0,Y 356.669,Z 383.986,A -85,B 0,C 180,E1 -13790.661,E2 -13790.661} C_VEL
LIN {X 0,Y 357.298,Z 370.943,A -85,B 0,C 180,E1 -13791.094,E2 -13791.094} C_VEL
LIN {X 0,Y 358.688,Z 300.601,A -85,B 0,C 180,E1 -13792.524,E2 -13792.524} C_VEL
LIN {X 0,Y 353.923,Z 274.293,A -85,B 0,C 180,E1 -13793.458,E2 -13793.458} C_VEL
LIN {X 0,Y 351.886,Z 264.746,A -85,B 0,C 180,E1 -13793.845,E2 -13793.845} C_VEL
LIN {X 0,Y 352.511,Z 258.436,A -85,B 0,C 180,E1 -13795.382,E2 -13795.382} C_VEL
LIN {X 0,Y 350.434,Z 247.552,A -85,B 0,C 180,E1 -13798.345,E2 -13798.345} C_VEL
LIN {X 0,Y 347.747,Z 236.168,A -85,B 0,C 180,E1 -13801.657,E2 -13801.657} C_VEL
LIN {X 0,Y 347.745,Z 236.167,A -85,B 0,C 180,E1 -13804.464,E2 -13804.464} C_VEL
LIN {X 0,Y 347.774,Z 236.165,A -85,B 0,C 180,E1 -13807.988,E2 -13807.988} C_VEL
LIN {X 0,Y 347.751,Z 236.169,A -85,B 0,C 180,E1 -13811.83,E2 -13811.83} C_VEL
LIN {X 0,Y 347.706,Z 236.173,A -85,B 0,C 180,E1 -13815.027,E2 -13815.027} C_VEL
LIN {X 0,Y 347.742,Z 236.167,A -85,B 0,C 180,E1 -13818.399,E2 -13818.399} C_VEL
LIN {X 0,Y 347.757,Z 236.163,A -85,B 0,C 180,E1 -13822.679,E2 -13822.679} C_VEL
LIN {X 0,Y 347.749,Z 236.162,A -85,B 0,C 180,E1 -13825.956,E2 -13825.956} C_VEL
LIN {X 0,Y 347.745,Z 236.163,A -85,B 0,C 180,E1 -13829.652,E2 -13829.652} C_VEL
LIN {X 0,Y 347.785,Z 236.159,A -85,B 0,C 180,E1 -13833.604,E2 -13833.604} C_VEL
LIN {X 0,Y 347.784,Z 236.162,A -85,B 0,C 180,E1 -13836.162,E2 -13836.162} C_VEL
LIN {X 0,Y 347.8,Z 236.161,A -85,B 0,C 180,E1 -13839.909,E2 -13839.909} C_VEL
LIN {X 0,Y 347.833,Z 236.152,A -85,B 0,C 180,E1 -13843.568,E2 -13843.568} C_VEL
LIN {X 0,Y 347.891,Z 236.147,A -85,B 0,C 180,E1 -13847.161,E2 -13847.161} C_VEL
LIN {X 0,Y 347.965,Z 236.138,A -85,B 0,C 180,E1 -13850.701,E2 -13850.701} C_VEL
LIN {X 0,Y 348.094,Z 236.116,A -85,B 0,C 180,E1 -13853.042,E2 -13853.042} C_VEL
LIN {X 0,Y 348.196,Z 236.103,A -85,B 0,C 180,E1 -13857.687,E2 -13857.687} C_VEL
LIN {X 0,Y 348.324,Z 236.094,A -85,B 0,C 180,E1 -13860,E2 -13860} C_VEL
LIN {X 0,Y 348.204,Z 236.103,A -85,B 0,C 180,E1 -13862.314,E2 -13862.314} C_VEL
LIN {X 0,Y 348.069,Z 236.127,A -85,B 0,C 180,E1 -13866.959,E2 -13866.959} C_VEL
LIN {X 0,Y 347.897,Z 236.147,A -85,B 0,C 180,E1 -13870.475,E2 -13870.475} C_VEL
LIN {X 0,Y 347.9,Z 236.143,A -85,B 0,C 180,E1 -13874.15,E2 -13874.15} C_VEL
LIN {X 0,Y 347.83,Z 236.148,A -85,B 0,C 180,E1 -13878.259,E2 -13878.259} C_VEL
LIN {X 0,Y 347.79,Z 236.156,A -85,B 0,C 180,E1 -13881.635,E2 -13881.635} C_VEL
LIN {X 0,Y 347.814,Z 236.16,A -85,B 0,C 180,E1 -13885.109,E2 -13885.109} C_VEL
LIN {X 0,Y 347.809,Z 236.161,A -85,B 0,C 180,E1 -13887.694,E2 -13887.694} C_VEL
LIN {X 0,Y 347.751,Z 236.162,A -85,B 0,C 180,E1 -13890.348,E2 -13890.348} C_VEL
LIN {X 0,Y 347.75,Z 236.167,A -85,B 0,C 180,E1 -13894.044,E2 -13894.044} C_VEL
LIN {X 0,Y 347.766,Z 236.166,A -85,B 0,C 180,E1 -13897.321,E2 -13897.321} C_VEL
LIN {X 0,Y 347.733,Z 236.169,A -85,B 0,C 180,E1 -13900.297,E2 -13900.297} C_VEL
LIN {X 0,Y 347.725,Z 236.172,A -85,B 0,C 180,E1 -13903.408,E2 -13903.408} C_VEL
LIN {X 0,Y 347.729,Z 236.163,A -85,B 0,C 180,E1 -13906.686,E2 -13906.686} C_VEL
LIN {X 0,Y 347.703,Z 236.171,A -85,B 0,C 180,E1 -13910.182,E2 -13910.182} C_VEL
LIN {X 0,Y 347.759,Z 236.171,A -85,B 0,C 180,E1 -13912.679,E2 -13912.679} C_VEL
LIN {X 0,Y 347.75,Z 236.17,A -85,B 0,C 180,E1 -13915.956,E2 -13915.956} C_VEL
LIN {X 0,Y 347.78,Z 236.306,A -85,B 0,C 180,E1 -13916.73,E2 -13916.73} C_VEL
LIN {X 0,Y 350.338,Z 247.485,A -85,B 0,C 180,E1 -13920.075,E2 -13920.075} C_VEL
LIN {X 0,Y 355.969,Z 261.655,A -85,B 0,C 180,E1 -13920.85,E2 -13920.85} C_VEL
LIN {X 0,Y 359.184,Z 276.068,A -85,B 0,C 180,E1 -13921.409,E2 -13921.409} C_VEL
LIN {X 0,Y 357.553,Z 355.055,A -85,B 0,C 180,E1 -13923.026,E2 -13923.026} C_VEL
LIN {X 0,Y 356.823,Z 368.723,A -85,B 0,C 180,E1 -13923.537,E2 -13923.537} C_VEL
LIN {X 0,Y 355.983,Z 381.418,A -85,B 0,C 180,E1 -13924.257,E2 -13924.257} C_VEL
LIN {X 0,Y 354.875,Z 392.645,A -85,B 0,C 180,E1 -13925.112,E2 -13925.112} C_VEL
LIN {X 0,Y 353.573,Z 404.319,A -85,B 0,C 180,E1 -13926.268,E2 -13926.268} C_VEL
LIN {X 0,Y 352.105,Z 414.746,A -85,B 0,C 180,E1 -13927.559,E2 -13927.559} C_VEL
LIN {X 0,Y 351.074,Z 423.271,A -85,B 0,C 180,E1 -13928.879,E2 -13928.879} C_VEL
LIN {X 0,Y 349.722,Z 432.439,A -85,B 0,C 180,E1 -13930.631,E2 -13930.631} C_VEL
LIN {X 0,Y 348.668,Z 439.83,A -85,B 0,C 180,E1 -13932.401,E2 -13932.401} C_VEL
LIN {X 0,Y 347.785,Z 445.713,A -85,B 0,C 180,E1 -13934.169,E2 -13934.169} C_VEL
LIN {X 0,Y 347.157,Z 450.326,A -85,B 0,C 180,E1 -13935.94,E2 -13935.94} C_VEL
LIN {X 0,Y 346.829,Z 452.755,A -85,B 0,C 180,E1 -13937.121,E2 -13937.121} C_VEL
LIN {X 0,Y 346.543,Z 454.732,A -85,B 0,C 180,E1 -13938.299,E2 -13938.299} C_VEL
LIN {X 0,Y 346.277,Z 456.292,A -85,B 0,C 180,E1 -13939.475,E2 -13939.475} C_VEL
LIN {X 0,Y 346.176,Z 457.417,A -85,B 0,C 180,E1 -13940.653,E2 -13940.653} C_VEL
LIN {X 0,Y 346.182,Z 458.425,A -85,B 0,C 180,E1 -13943.003,E2 -13943.003} C_VEL
LIN {X 0,Y 346.182,Z 458.355,A -85,B 0,C 180,E1 -13944.174,E2 -13944.174} C_VEL
LIN {X 0,Y 346.166,Z 457.878,A -85,B 0,C 180,E1 -13945.342,E2 -13945.342} C_VEL
LIN {X 0,Y 346.157,Z 456.983,A -85,B 0,C 180,E1 -13946.508,E2 -13946.508} C_VEL
LIN {X 0,Y 346.325,Z 454.017,A -85,B 0,C 180,E1 -13948.837,E2 -13948.837} C_VEL
LIN {X 0,Y 346.527,Z 450.642,A -85,B 0,C 180,E1 -13950.581,E2 -13950.581} C_VEL
LIN {X 0,Y 346.868,Z 446.201,A -85,B 0,C 180,E1 -13952.322,E2 -13952.322} C_VEL
LIN {X 0,Y 347.57,Z 439.469,A -85,B 0,C 180,E1 -13954.349,E2 -13954.349} C_VEL
LIN {X 0,Y 348.28,Z 432.163,A -85,B 0,C 180,E1 -13956.081,E2 -13956.081} C_VEL
LIN {X 0,Y 349.354,Z 423.081,A -85,B 0,C 180,E1 -13957.804,E2 -13957.804} C_VEL
LIN {X 0,Y 350.481,Z 412.588,A -85,B 0,C 180,E1 -13959.377,E2 -13959.377} C_VEL
LIN {X 0,Y 351.536,Z 401.912,A -85,B 0,C 180,E1 -13960.657,E2 -13960.657} C_VEL
LIN {X 0,Y 352.402,Z 391.553,A -85,B 0,C 180,E1 -13961.649,E2 -13961.649} C_VEL
LIN {X 0,Y 353.212,Z 380.232,A -85,B 0,C 180,E1 -13962.497,E2 -13962.497} C_VEL
LIN {X 0,Y 353.899,Z 366.937,A -85,B 0,C 180,E1 -13963.229,E2 -13963.229} C_VEL
LIN {X 0,Y 354.305,Z 354.564,A -85,B 0,C 180,E1 -13963.684,E2 -13963.684} C_VEL
LIN {X 0,Y 355.766,Z 274.429,A -85,B 0,C 180,E1 -13965.308,E2 -13965.308} C_VEL
LIN {X 0,Y 353.377,Z 260.618,A -85,B 0,C 180,E1 -13965.735,E2 -13965.735} C_VEL
LIN {X 0,Y 351.998,Z 256.851,A -85,B 0,C 180,E1 -13965.896,E2 -13965.896} C_VEL
LIN {X 0,Y 349.703,Z 253.57,A -85,B 0,C 180,E1 -13966.1,E2 -13966.1} C_VEL
LIN {X 0,Y 346.149,Z 249.821,A -85,B 0,C 180,E1 -13966.441,E2 -13966.441} C_VEL
LIN {X 0,Y 343.794,Z 247.32,A -85,B 0,C 180,E1 -13966.815,E2 -13966.815} C_VEL
LIN {X 0,Y 342.564,Z 245.433,A -85,B 0,C 180,E1 -13967.229,E2 -13967.229} C_VEL
LIN {X 0,Y 342.45,Z 245.089,A -85,B 0,C 180,E1 -13967.324,E2 -13967.324} C_VEL
LIN {X 0,Y 340.786,Z 237.037,A -85,B 0,C 180,E1 -13969.658,E2 -13969.658} C_VEL
LIN {X 0,Y 340.723,Z 237.043,A -85,B 0,C 180,E1 -13973.073,E2 -13973.073} C_VEL
LIN {X 0,Y 340.747,Z 237.037,A -85,B 0,C 180,E1 -13975.666,E2 -13975.666} C_VEL
LIN {X 0,Y 340.734,Z 237.038,A -85,B 0,C 180,E1 -13979.671,E2 -13979.671} C_VEL
LIN {X 0,Y 340.694,Z 237.043,A -85,B 0,C 180,E1 -13983.846,E2 -13983.846} C_VEL
LIN {X 0,Y 340.707,Z 237.047,A -85,B 0,C 180,E1 -13986.741,E2 -13986.741} C_VEL
LIN {X 0,Y 340.69,Z 237.046,A -85,B 0,C 180,E1 -13990.247,E2 -13990.247} C_VEL
LIN {X 0,Y 340.669,Z 237.046,A -85,B 0,C 180,E1 -13993.776,E2 -13993.776} C_VEL
LIN {X 0,Y 340.677,Z 237.047,A -85,B 0,C 180,E1 -13997.095,E2 -13997.095} C_VEL
LIN {X 0,Y 340.699,Z 237.045,A -85,B 0,C 180,E1 -14000.247,E2 -14000.247} C_VEL
LIN {X 0,Y 340.711,Z 237.041,A -85,B 0,C 180,E1 -14003.559,E2 -14003.559} C_VEL
LIN {X 0,Y 340.693,Z 237.044,A -85,B 0,C 180,E1 -14006.153,E2 -14006.153} C_VEL
LIN {X 0,Y 340.742,Z 237.039,A -85,B 0,C 180,E1 -14010.329,E2 -14010.329} C_VEL
LIN {X 0,Y 340.804,Z 237.032,A -85,B 0,C 180,E1 -14013.02,E2 -14013.02} C_VEL
LIN {X 0,Y 340.73,Z 237.039,A -85,B 0,C 180,E1 -14016.927,E2 -14016.927} C_VEL
LIN {X 0,Y 340.791,Z 237.036,A -85,B 0,C 180,E1 -14020.733,E2 -14020.733} C_VEL
LIN {X 0,Y 340.787,Z 237.032,A -85,B 0,C 180,E1 -14023.218,E2 -14023.218} C_VEL
LIN {X 0,Y 340.845,Z 237.026,A -85,B 0,C 180,E1 -14026.89,E2 -14026.89} C_VEL
LIN {X 0,Y 340.882,Z 237.022,A -85,B 0,C 180,E1 -14030.506,E2 -14030.506} C_VEL
LIN {X 0,Y 341.025,Z 237.003,A -85,B 0,C 180,E1 -14034.085,E2 -14034.085} C_VEL
LIN {X 0,Y 341.168,Z 236.983,A -85,B 0,C 180,E1 -14037.639,E2 -14037.639} C_VEL
LIN {X 0,Y 341.275,Z 236.972,A -85,B 0,C 180,E1 -14040,E2 -14040} C_VEL
LIN {X 0,Y 341.165,Z 236.988,A -85,B 0,C 180,E1 -14042.361,E2 -14042.361} C_VEL
LIN {X 0,Y 341.076,Z 236.997,A -85,B 0,C 180,E1 -14047.102,E2 -14047.102} C_VEL
LIN {X 0,Y 340.871,Z 237.025,A -85,B 0,C 180,E1 -14050.694,E2 -14050.694} C_VEL
LIN {X 0,Y 340.863,Z 237.025,A -85,B 0,C 180,E1 -14054.325,E2 -14054.325} C_VEL
LIN {X 0,Y 340.786,Z 237.036,A -85,B 0,C 180,E1 -14058.44,E2 -14058.44} C_VEL
LIN {X 0,Y 340.718,Z 237.041,A -85,B 0,C 180,E1 -14061.842,E2 -14061.842} C_VEL
LIN {X 0,Y 340.751,Z 237.039,A -85,B 0,C 180,E1 -14064.838,E2 -14064.838} C_VEL
LIN {X 0,Y 340.685,Z 237.048,A -85,B 0,C 180,E1 -14068.325,E2 -14068.325} C_VEL
LIN {X 0,Y 340.694,Z 237.045,A -85,B 0,C 180,E1 -14071.045,E2 -14071.045} C_VEL
LIN {X 0,Y 340.718,Z 237.04,A -85,B 0,C 180,E1 -14075.279,E2 -14075.279} C_VEL
LIN {X 0,Y 340.694,Z 237.048,A -85,B 0,C 180,E1 -14078.383,E2 -14078.383} C_VEL
LIN {X 0,Y 340.694,Z 237.045,A -85,B 0,C 180,E1 -14082.045,E2 -14082.045} C_VEL
LIN {X 0,Y 340.652,Z 237.051,A -85,B 0,C 180,E1 -14086.227,E2 -14086.227} C_VEL
LIN {X 0,Y 340.685,Z 237.044,A -85,B 0,C 180,E1 -14089.754,E2 -14089.754} C_VEL
LIN {X 0,Y 340.707,Z 237.042,A -85,B 0,C 180,E1 -14093.259,E2 -14093.259} C_VEL
LIN {X 0,Y 340.693,Z 237.046,A -85,B 0,C 180,E1 -14096.154,E2 -14096.154} C_VEL
LIN {X 0,Y 340.76,Z 237.232,A -85,B 0,C 180,E1 -14100.24,E2 -14100.24} C_VEL
LIN {X 0,Y 343.027,Z 248.13,A -85,B 0,C 180,E1 -14103.209,E2 -14103.209} C_VEL
LIN {X 0,Y 344.236,Z 255.978,A -85,B 0,C 180,E1 -14105.258,E2 -14105.258} C_VEL
LIN {X 0,Y 343.37,Z 264.8,A -85,B 0,C 180,E1 -14107.392,E2 -14107.392} C_VEL
LIN {X 0,Y 348.589,Z 299.863,A -85,B 0,C 180,E1 -14108.473,E2 -14108.473} C_VEL
LIN {X 0,Y 347.401,Z 373.182,A -85,B 0,C 180,E1 -14110,E2 -14110} C_VEL
LIN {X 0,Y 346.709,Z 386.473,A -85,B 0,C 180,E1 -14110.499,E2 -14110.499} C_VEL
LIN {X 0,Y 345.908,Z 398.669,A -85,B 0,C 180,E1 -14111.183,E2 -14111.183} C_VEL
LIN {X 0,Y 344.944,Z 410.146,A -85,B 0,C 180,E1 -14112.052,E2 -14112.052} C_VEL
LIN {X 0,Y 343.768,Z 421.924,A -85,B 0,C 180,E1 -14113.216,E2 -14113.216} C_VEL
LIN {X 0,Y 342.602,Z 433.039,A -85,B 0,C 180,E1 -14114.61,E2 -14114.61} C_VEL
LIN {X 0,Y 341.725,Z 442.022,A -85,B 0,C 180,E1 -14116.016,E2 -14116.016} C_VEL
LIN {X 0,Y 340.917,Z 449.813,A -85,B 0,C 180,E1 -14117.499,E2 -14117.499} C_VEL
LIN {X 0,Y 340.112,Z 457.423,A -85,B 0,C 180,E1 -14119.282,E2 -14119.282} C_VEL
LIN {X 0,Y 339.598,Z 463.542,A -85,B 0,C 180,E1 -14121.071,E2 -14121.071} C_VEL
LIN {X 0,Y 339.27,Z 468.384,A -85,B 0,C 180,E1 -14122.86,E2 -14122.86} C_VEL
LIN {X 0,Y 339.096,Z 471.945,A -85,B 0,C 180,E1 -14124.566,E2 -14124.566} C_VEL
LIN {X 0,Y 339.071,Z 474.779,A -85,B 0,C 180,E1 -14126.435,E2 -14126.435} C_VEL
LIN {X 0,Y 339.019,Z 476.903,A -85,B 0,C 180,E1 -14128.812,E2 -14128.812} C_VEL
LIN {X 0,Y 339.067,Z 477.328,A -85,B 0,C 180,E1 -14130,E2 -14130} C_VEL
LIN {X 0,Y 338.996,Z 477.003,A -85,B 0,C 180,E1 -14132.376,E2 -14132.376} C_VEL
LIN {X 0,Y 339.065,Z 476.265,A -85,B 0,C 180,E1 -14133.565,E2 -14133.565} C_VEL
LIN {X 0,Y 339.134,Z 473.587,A -85,B 0,C 180,E1 -14135.889,E2 -14135.889} C_VEL
LIN {X 0,Y 339.408,Z 470.318,A -85,B 0,C 180,E1 -14137.735,E2 -14137.735} C_VEL
LIN {X 0,Y 339.911,Z 466.088,A -85,B 0,C 180,E1 -14139.521,E2 -14139.521} C_VEL
LIN {X 0,Y 340.735,Z 459.682,A -85,B 0,C 180,E1 -14141.602,E2 -14141.602} C_VEL
LIN {X 0,Y 341.85,Z 452.707,A -85,B 0,C 180,E1 -14143.373,E2 -14143.373} C_VEL
LIN {X 0,Y 343.125,Z 443.987,A -85,B 0,C 180,E1 -14145.138,E2 -14145.138} C_VEL
LIN {X 0,Y 344.332,Z 435.077,A -85,B 0,C 180,E1 -14146.604,E2 -14146.604} C_VEL
LIN {X 0,Y 345.731,Z 425.296,A -85,B 0,C 180,E1 -14147.906,E2 -14147.906} C_VEL
LIN {X 0,Y 347.137,Z 414.548,A -85,B 0,C 180,E1 -14149.054,E2 -14149.054} C_VEL
LIN {X 0,Y 348.304,Z 404.476,A -85,B 0,C 180,E1 -14149.907,E2 -14149.907} C_VEL
LIN {X 0,Y 349.44,Z 392.516,A -85,B 0,C 180,E1 -14150.684,E2 -14150.684} C_VEL
LIN {X 0,Y 350.353,Z 379.677,A -85,B 0,C 180,E1 -14151.278,E2 -14151.278} C_VEL
LIN {X 0,Y 350.99,Z 366.607,A -85,B 0,C 180,E1 -14151.646,E2 -14151.646} C_VEL
LIN {X 0,Y 352.241,Z 301.513,A -85,B 0,C 180,E1 -14152.986,E2 -14152.986} C_VEL
LIN {X 0,Y 347.69,Z 276.259,A -85,B 0,C 180,E1 -14153.906,E2 -14153.906} C_VEL
LIN {X 0,Y 345.205,Z 264.584,A -85,B 0,C 180,E1 -14154.38,E2 -14154.38} C_VEL
LIN {X 0,Y 345.612,Z 259.883,A -85,B 0,C 180,E1 -14155.555,E2 -14155.555} C_VEL
LIN {X 0,Y 343.384,Z 248.147,A -85,B 0,C 180,E1 -14158.828,E2 -14158.828} C_VEL
LIN {X 0,Y 340.688,Z 237.048,A -85,B 0,C 180,E1 -14162.137,E2 -14162.137} C_VEL
LIN {X 0,Y 340.719,Z 237.042,A -85,B 0,C 180,E1 -14165.279,E2 -14165.279} C_VEL
LIN {X 0,Y 340.71,Z 237.044,A -85,B 0,C 180,E1 -14168.386,E2 -14168.386} C_VEL
LIN {X 0,Y 340.699,Z 237.047,A -85,B 0,C 180,E1 -14172.045,E2 -14172.045} C_VEL
LIN {X 0,Y 340.652,Z 237.051,A -85,B 0,C 180,E1 -14176.227,E2 -14176.227} C_VEL
LIN {X 0,Y 340.672,Z 237.048,A -85,B 0,C 180,E1 -14178.688,E2 -14178.688} C_VEL
LIN {X 0,Y 340.719,Z 237.042,A -85,B 0,C 180,E1 -14181.771,E2 -14181.771} C_VEL
LIN {X 0,Y 340.723,Z 237.04,A -85,B 0,C 180,E1 -14185.595,E2 -14185.595} C_VEL
LIN {X 0,Y 340.696,Z 237.045,A -85,B 0,C 180,E1 -14188.955,E2 -14188.955} C_VEL
LIN {X 0,Y 340.711,Z 237.042,A -85,B 0,C 180,E1 -14192.496,E2 -14192.496} C_VEL
LIN {X 0,Y 340.752,Z 237.038,A -85,B 0,C 180,E1 -14195.638,E2 -14195.638} C_VEL
LIN {X 0,Y 340.73,Z 237.038,A -85,B 0,C 180,E1 -14199.473,E2 -14199.473} C_VEL
LIN {X 0,Y 340.793,Z 237.031,A -85,B 0,C 180,E1 -14201.981,E2 -14201.981} C_VEL
LIN {X 0,Y 340.87,Z 237.025,A -85,B 0,C 180,E1 -14205.705,E2 -14205.705} C_VEL
LIN {X 0,Y 340.871,Z 237.02,A -85,B 0,C 180,E1 -14209.306,E2 -14209.306} C_VEL
LIN {X 0,Y 341.062,Z 236.992,A -85,B 0,C 180,E1 -14212.898,E2 -14212.898} C_VEL
LIN {X 0,Y 341.157,Z 236.98,A -85,B 0,C 180,E1 -14217.639,E2 -14217.639} C_VEL
LIN {X 0,Y 341.275,Z 236.972,A -85,B 0,C 180,E1 -14220,E2 -14220} C_VEL
LIN {X 0,Y 341.165,Z 236.98,A -85,B 0,C 180,E1 -14222.361,E2 -14222.361} C_VEL
LIN {X 0,Y 341.017,Z 237.005,A -85,B 0,C 180,E1 -14227.103,E2 -14227.103} C_VEL
LIN {X 0,Y 340.849,Z 237.025,A -85,B 0,C 180,E1 -14230.695,E2 -14230.695} C_VEL
LIN {X 0,Y 340.864,Z 237.019,A -85,B 0,C 180,E1 -14234.325,E2 -14234.325} C_VEL
LIN {X 0,Y 340.787,Z 237.025,A -85,B 0,C 180,E1 -14238.441,E2 -14238.441} C_VEL
LIN {X 0,Y 340.755,Z 237.03,A -85,B 0,C 180,E1 -14241.857,E2 -14241.857} C_VEL
LIN {X 0,Y 340.773,Z 237.031,A -85,B 0,C 180,E1 -14245.665,E2 -14245.665} C_VEL
LIN {X 0,Y 340.73,Z 237.04,A -85,B 0,C 180,E1 -14248.321,E2 -14248.321} C_VEL
LIN {X 0,Y 340.699,Z 237.043,A -85,B 0,C 180,E1 -14251.045,E2 -14251.045} C_VEL
LIN {X 0,Y 340.72,Z 237.046,A -85,B 0,C 180,E1 -14255.279,E2 -14255.279} C_VEL
LIN {X 0,Y 340.712,Z 237.042,A -85,B 0,C 180,E1 -14258.386,E2 -14258.386} C_VEL
LIN {X 0,Y 340.7,Z 237.046,A -85,B 0,C 180,E1 -14262.046,E2 -14262.046} C_VEL
LIN {X 0,Y 340.685,Z 237.047,A -85,B 0,C 180,E1 -14265.462,E2 -14265.462} C_VEL
LIN {X 0,Y 340.673,Z 237.054,A -85,B 0,C 180,E1 -14268.689,E2 -14268.689} C_VEL
LIN {X 0,Y 340.721,Z 237.05,A -85,B 0,C 180,E1 -14271.771,E2 -14271.771} C_VEL
LIN {X 0,Y 340.725,Z 237.046,A -85,B 0,C 180,E1 -14275.596,E2 -14275.596} C_VEL
LIN {X 0,Y 340.724,Z 237.183,A -85,B 0,C 180,E1 -14276.246,E2 -14276.246} C_VEL
LIN {X 0,Y 343.155,Z 247.676,A -85,B 0,C 180,E1 -14279.472,E2 -14279.472} C_VEL
LIN {X 0,Y 349.755,Z 263.823,A -85,B 0,C 180,E1 -14280.408,E2 -14280.408} C_VEL
LIN {X 0,Y 352.848,Z 277.909,A -85,B 0,C 180,E1 -14280.966,E2 -14280.966} C_VEL
LIN {X 0,Y 351.018,Z 355.699,A -85,B 0,C 180,E1 -14282.581,E2 -14282.581} C_VEL
LIN {X 0,Y 350.275,Z 369.65,A -85,B 0,C 180,E1 -14283.123,E2 -14283.123} C_VEL
LIN {X 0,Y 349.322,Z 382.612,A -85,B 0,C 180,E1 -14283.89,E2 -14283.89} C_VEL
LIN {X 0,Y 347.977,Z 395.215,A -85,B 0,C 180,E1 -14284.904,E2 -14284.904} C_VEL
LIN {X 0,Y 346.687,Z 406.419,A -85,B 0,C 180,E1 -14286.081,E2 -14286.081} C_VEL
LIN {X 0,Y 345.309,Z 415.448,A -85,B 0,C 180,E1 -14287.25,E2 -14287.25} C_VEL
LIN {X 0,Y 344.108,Z 424.698,A -85,B 0,C 180,E1 -14288.745,E2 -14288.745} C_VEL
LIN {X 0,Y 342.911,Z 432.303,A -85,B 0,C 180,E1 -14290.235,E2 -14290.235} C_VEL
LIN {X 0,Y 341.782,Z 439.734,A -85,B 0,C 180,E1 -14292.035,E2 -14292.035} C_VEL
LIN {X 0,Y 340.841,Z 445.673,A -85,B 0,C 180,E1 -14293.837,E2 -14293.837} C_VEL
LIN {X 0,Y 340.164,Z 450.34,A -85,B 0,C 180,E1 -14295.645,E2 -14295.645} C_VEL
LIN {X 0,Y 339.644,Z 453.879,A -85,B 0,C 180,E1 -14297.451,E2 -14297.451} C_VEL
LIN {X 0,Y 339.226,Z 456.395,A -85,B 0,C 180,E1 -14299.254,E2 -14299.254} C_VEL
LIN {X 0,Y 339.113,Z 457.56,A -85,B 0,C 180,E1 -14300.456,E2 -14300.456} C_VEL
LIN {X 0,Y 339.092,Z 458.612,A -85,B 0,C 180,E1 -14302.856,E2 -14302.856} C_VEL
LIN {X 0,Y 339.083,Z 458.542,A -85,B 0,C 180,E1 -14304.198,E2 -14304.198} C_VEL
LIN {X 0,Y 339.08,Z 457.252,A -85,B 0,C 180,E1 -14306.435,E2 -14306.435} C_VEL
LIN {X 0,Y 339.221,Z 454.33,A -85,B 0,C 180,E1 -14308.813,E2 -14308.813} C_VEL
LIN {X 0,Y 339.452,Z 450.998,A -85,B 0,C 180,E1 -14310.593,E2 -14310.593} C_VEL
LIN {X 0,Y 339.804,Z 446.605,A -85,B 0,C 180,E1 -14312.371,E2 -14312.371} C_VEL
LIN {X 0,Y 340.507,Z 439.954,A -85,B 0,C 180,E1 -14314.439,E2 -14314.439} C_VEL
LIN {X 0,Y 341.254,Z 432.708,A -85,B 0,C 180,E1 -14316.207,E2 -14316.207} C_VEL
LIN {X 0,Y 342.363,Z 423.712,A -85,B 0,C 180,E1 -14317.965,E2 -14317.965} C_VEL
LIN {X 0,Y 343.527,Z 413.335,A -85,B 0,C 180,E1 -14319.568,E2 -14319.568} C_VEL
LIN {X 0,Y 344.595,Z 402.774,A -85,B 0,C 180,E1 -14320.874,E2 -14320.874} C_VEL
LIN {X 0,Y 345.652,Z 390.914,A -85,B 0,C 180,E1 -14322.029,E2 -14322.029} C_VEL
LIN {X 0,Y 346.517,Z 379.339,A -85,B 0,C 180,E1 -14322.891,E2 -14322.891} C_VEL
LIN {X 0,Y 347.158,Z 366.151,A -85,B 0,C 180,E1 -14323.616,E2 -14323.616} C_VEL
LIN {X 0,Y 347.602,Z 352.981,A -85,B 0,C 180,E1 -14324.079,E2 -14324.079} C_VEL
LIN {X 0,Y 349.004,Z 274.867,A -85,B 0,C 180,E1 -14325.685,E2 -14325.685} C_VEL
LIN {X 0,Y 345.175,Z 254.125,A -85,B 0,C 180,E1 -14326.361,E2 -14326.361} C_VEL
LIN {X 0,Y 342.853,Z 247.402,A -85,B 0,C 180,E1 -14326.677,E2 -14326.677} C_VEL
LIN {X 0,Y 342.45,Z 245.089,A -85,B 0,C 180,E1 -14327.324,E2 -14327.324} C_VEL
LIN {X 0,Y 341.274,Z 243.363,A -85,B 0,C 180,E1 -14327.885,E2 -14327.885} C_VEL
LIN {X 0,Y 334.503,Z 238.683,A -85,B 0,C 180,E1 -14329.719,E2 -14329.719} C_VEL
LIN {X 0,Y 333.734,Z 237.947,A -85,B 0,C 180,E1 -14330.267,E2 -14330.267} C_VEL
LIN {X 0,Y 333.701,Z 237.919,A -85,B 0,C 180,E1 -14330.382,E2 -14330.382} C_VEL
LIN {X 0,Y 333.67,Z 237.919,A -85,B 0,C 180,E1 -14333.59,E2 -14333.59} C_VEL
LIN {X 0,Y 333.678,Z 237.92,A -85,B 0,C 180,E1 -14336.251,E2 -14336.251} C_VEL
LIN {X 0,Y 333.662,Z 237.923,A -85,B 0,C 180,E1 -14340.366,E2 -14340.366} C_VEL
LIN {X 0,Y 333.639,Z 237.924,A -85,B 0,C 180,E1 -14343.208,E2 -14343.208} C_VEL
LIN {X 0,Y 333.678,Z 237.919,A -85,B 0,C 180,E1 -14346.139,E2 -14346.139} C_VEL
LIN {X 0,Y 333.648,Z 237.922,A -85,B 0,C 180,E1 -14349.192,E2 -14349.192} C_VEL
LIN {X 0,Y 333.635,Z 237.927,A -85,B 0,C 180,E1 -14352.5,E2 -14352.5} C_VEL
LIN {X 0,Y 333.621,Z 237.925,A -85,B 0,C 180,E1 -14355.959,E2 -14355.959} C_VEL
LIN {X 0,Y 333.647,Z 237.922,A -85,B 0,C 180,E1 -14359.315,E2 -14359.315} C_VEL
LIN {X 0,Y 333.666,Z 237.92,A -85,B 0,C 180,E1 -14363.168,E2 -14363.168} C_VEL
LIN {X 0,Y 333.675,Z 237.917,A -85,B 0,C 180,E1 -14365.341,E2 -14365.341} C_VEL
LIN {X 0,Y 333.691,Z 237.914,A -85,B 0,C 180,E1 -14369.637,E2 -14369.637} C_VEL
LIN {X 0,Y 333.74,Z 237.913,A -85,B 0,C 180,E1 -14372.401,E2 -14372.401} C_VEL
LIN {X 0,Y 333.727,Z 237.911,A -85,B 0,C 180,E1 -14375.09,E2 -14375.09} C_VEL
LIN {X 0,Y 333.686,Z 237.916,A -85,B 0,C 180,E1 -14379.019,E2 -14379.019} C_VEL
LIN {X 0,Y 333.794,Z 237.902,A -85,B 0,C 180,E1 -14381.589,E2 -14381.589} C_VEL
LIN {X 0,Y 333.809,Z 237.9,A -85,B 0,C 180,E1 -14385.576,E2 -14385.576} C_VEL
LIN {X 0,Y 333.818,Z 237.897,A -85,B 0,C 180,E1 -14389.077,E2 -14389.077} C_VEL
LIN {X 0,Y 333.963,Z 237.886,A -85,B 0,C 180,E1 -14392.746,E2 -14392.746} C_VEL
LIN {X 0,Y 333.802,Z 237.903,A -85,B 0,C 180,E1 -14395.169,E2 -14395.169} C_VEL
LIN {X 0,Y 334.105,Z 237.863,A -85,B 0,C 180,E1 -14397.589,E2 -14397.589} C_VEL
LIN {X 0,Y 334.226,Z 237.85,A -85,B 0,C 180,E1 -14400,E2 -14400} C_VEL
LIN {X 0,Y 334.102,Z 237.868,A -85,B 0,C 180,E1 -14402.411,E2 -14402.411} C_VEL
LIN {X 0,Y 334.026,Z 237.875,A -85,B 0,C 180,E1 -14407.252,E2 -14407.252} C_VEL
LIN {X 0,Y 333.834,Z 237.899,A -85,B 0,C 180,E1 -14410.922,E2 -14410.922} C_VEL
LIN {X 0,Y 333.808,Z 237.907,A -85,B 0,C 180,E1 -14414.634,E2 -14414.634} C_VEL
LIN {X 0,Y 333.724,Z 237.916,A -85,B 0,C 180,E1 -14418.618,E2 -14418.618} C_VEL
LIN {X 0,Y 333.655,Z 237.923,A -85,B 0,C 180,E1 -14422.281,E2 -14422.281} C_VEL
LIN {X 0,Y 333.7,Z 237.915,A -85,B 0,C 180,E1 -14425.094,E2 -14425.094} C_VEL
LIN {X 0,Y 333.655,Z 237.922,A -85,B 0,C 180,E1 -14428.977,E2 -14428.977} C_VEL
LIN {X 0,Y 333.643,Z 237.928,A -85,B 0,C 180,E1 -14432.587,E2 -14432.587} C_VEL
LIN {X 0,Y 333.675,Z 237.919,A -85,B 0,C 180,E1 -14436.139,E2 -14436.139} C_VEL
LIN {X 0,Y 333.62,Z 237.925,A -85,B 0,C 180,E1 -14439.196,E2 -14439.196} C_VEL
LIN {X 0,Y 333.629,Z 237.929,A -85,B 0,C 180,E1 -14442.499,E2 -14442.499} C_VEL
LIN {X 0,Y 333.596,Z 237.928,A -85,B 0,C 180,E1 -14445.955,E2 -14445.955} C_VEL
LIN {X 0,Y 333.646,Z 237.921,A -85,B 0,C 180,E1 -14449.316,E2 -14449.316} C_VEL
LIN {X 0,Y 333.667,Z 237.92,A -85,B 0,C 180,E1 -14453.168,E2 -14453.168} C_VEL
LIN {X 0,Y 333.638,Z 237.927,A -85,B 0,C 180,E1 -14456.792,E2 -14456.792} C_VEL
LIN {X 0,Y 333.697,Z 238.03,A -85,B 0,C 180,E1 -14459.88,E2 -14459.88} C_VEL
LIN {X 0,Y 335.999,Z 248.988,A -85,B 0,C 180,E1 -14462.939,E2 -14462.939} C_VEL
LIN {X 0,Y 337.286,Z 256.843,A -85,B 0,C 180,E1 -14465.042,E2 -14465.042} C_VEL
LIN {X 0,Y 336.494,Z 264.606,A -85,B 0,C 180,E1 -14466.96,E2 -14466.96} C_VEL
LIN {X 0,Y 341.022,Z 294.41,A -85,B 0,C 180,E1 -14467.915,E2 -14467.915} C_VEL
LIN {X 0,Y 341.943,Z 302.545,A -85,B 0,C 180,E1 -14468.147,E2 -14468.147} C_VEL
LIN {X 0,Y 340.627,Z 373.788,A -85,B 0,C 180,E1 -14469.664,E2 -14469.664} C_VEL
LIN {X 0,Y 339.905,Z 386.812,A -85,B 0,C 180,E1 -14470.171,E2 -14470.171} C_VEL
LIN {X 0,Y 339.082,Z 398.87,A -85,B 0,C 180,E1 -14470.868,E2 -14470.868} C_VEL
LIN {X 0,Y 337.992,Z 411.035,A -85,B 0,C 180,E1 -14471.826,E2 -14471.826} C_VEL
LIN {X 0,Y 336.8,Z 422.606,A -85,B 0,C 180,E1 -14473.014,E2 -14473.014} C_VEL
LIN {X 0,Y 335.631,Z 433.393,A -85,B 0,C 180,E1 -14474.413,E2 -14474.413} C_VEL
LIN {X 0,Y 334.8,Z 441.548,A -85,B 0,C 180,E1 -14475.721,E2 -14475.721} C_VEL
LIN {X 0,Y 333.93,Z 449.392,A -85,B 0,C 180,E1 -14477.233,E2 -14477.233} C_VEL
LIN {X 0,Y 333.078,Z 457.044,A -85,B 0,C 180,E1 -14479.053,E2 -14479.053} C_VEL
LIN {X 0,Y 332.552,Z 463.199,A -85,B 0,C 180,E1 -14480.88,E2 -14480.88} C_VEL
LIN {X 0,Y 332.195,Z 468.073,A -85,B 0,C 180,E1 -14482.707,E2 -14482.707} C_VEL
LIN {X 0,Y 332.062,Z 471.089,A -85,B 0,C 180,E1 -14484.124,E2 -14484.124} C_VEL
LIN {X 0,Y 331.996,Z 474.525,A -85,B 0,C 180,E1 -14486.359,E2 -14486.359} C_VEL
LIN {X 0,Y 331.924,Z 476.679,A -85,B 0,C 180,E1 -14488.787,E2 -14488.787} C_VEL
LIN {X 0,Y 331.97,Z 477.125,A -85,B 0,C 180,E1 -14490,E2 -14490} C_VEL
LIN {X 0,Y 331.914,Z 476.826,A -85,B 0,C 180,E1 -14492.427,E2 -14492.427} C_VEL
LIN {X 0,Y 331.969,Z 476.101,A -85,B 0,C 180,E1 -14493.641,E2 -14493.641} C_VEL
LIN {X 0,Y 332.06,Z 473.671,A -85,B 0,C 180,E1 -14495.873,E2 -14495.873} C_VEL
LIN {X 0,Y 332.366,Z 470.221,A -85,B 0,C 180,E1 -14497.9,E2 -14497.9} C_VEL
LIN {X 0,Y 332.872,Z 466.02,A -85,B 0,C 180,E1 -14499.724,E2 -14499.724} C_VEL
LIN {X 0,Y 333.735,Z 459.648,A -85,B 0,C 180,E1 -14501.848,E2 -14501.848} C_VEL
LIN {X 0,Y 334.935,Z 452.719,A -85,B 0,C 180,E1 -14503.654,E2 -14503.654} C_VEL
LIN {X 0,Y 336.248,Z 444.054,A -85,B 0,C 180,E1 -14505.456,E2 -14505.456} C_VEL
LIN {X 0,Y 337.535,Z 435.196,A -85,B 0,C 180,E1 -14506.948,E2 -14506.948} C_VEL
LIN {X 0,Y 338.994,Z 425.48,A -85,B 0,C 180,E1 -14508.275,E2 -14508.275} C_VEL
LIN {X 0,Y 340.465,Z 414.846,A -85,B 0,C 180,E1 -14509.442,E2 -14509.442} C_VEL
LIN {X 0,Y 341.672,Z 404.893,A -85,B 0,C 180,E1 -14510.311,E2 -14510.311} C_VEL
LIN {X 0,Y 342.839,Z 393.168,A -85,B 0,C 180,E1 -14511.102,E2 -14511.102} C_VEL
LIN {X 0,Y 343.836,Z 379.742,A -85,B 0,C 180,E1 -14511.742,E2 -14511.742} C_VEL
LIN {X 0,Y 344.517,Z 366.62,A -85,B 0,C 180,E1 -14512.121,E2 -14512.121} C_VEL
LIN {X 0,Y 345.753,Z 302.27,A -85,B 0,C 180,E1 -14513.474,E2 -14513.474} C_VEL
LIN {X 0,Y 341.438,Z 278.022,A -85,B 0,C 180,E1 -14514.381,E2 -14514.381} C_VEL
LIN {X 0,Y 338.538,Z 264.381,A -85,B 0,C 180,E1 -14514.948,E2 -14514.948} C_VEL
LIN {X 0,Y 338.676,Z 260.966,A -85,B 0,C 180,E1 -14515.835,E2 -14515.835} C_VEL
LIN {X 0,Y 336.495,Z 249.717,A -85,B 0,C 180,E1 -14519.051,E2 -14519.051} C_VEL
LIN {X 0,Y 333.653,Z 237.924,A -85,B 0,C 180,E1 -14522.659,E2 -14522.659} C_VEL
LIN {X 0,Y 333.677,Z 237.92,A -85,B 0,C 180,E1 -14526.139,E2 -14526.139} C_VEL
LIN {X 0,Y 333.647,Z 237.927,A -85,B 0,C 180,E1 -14529.192,E2 -14529.192} C_VEL
LIN {X 0,Y 333.633,Z 237.926,A -85,B 0,C 180,E1 -14532.5,E2 -14532.5} C_VEL
LIN {X 0,Y 333.596,Z 237.931,A -85,B 0,C 180,E1 -14535.955,E2 -14535.955} C_VEL
LIN {X 0,Y 333.603,Z 237.931,A -85,B 0,C 180,E1 -14539.324,E2 -14539.324} C_VEL
LIN {X 0,Y 333.663,Z 237.917,A -85,B 0,C 180,E1 -14543.168,E2 -14543.168} C_VEL
LIN {X 0,Y 333.674,Z 237.921,A -85,B 0,C 180,E1 -14545.341,E2 -14545.341} C_VEL
LIN {X 0,Y 333.63,Z 237.924,A -85,B 0,C 180,E1 -14548.222,E2 -14548.222} C_VEL
LIN {X 0,Y 333.67,Z 237.914,A -85,B 0,C 180,E1 -14551.024,E2 -14551.024} C_VEL
LIN {X 0,Y 333.714,Z 237.909,A -85,B 0,C 180,E1 -14555.09,E2 -14555.09} C_VEL
LIN {X 0,Y 333.671,Z 237.914,A -85,B 0,C 180,E1 -14559.019,E2 -14559.019} C_VEL
LIN {X 0,Y 333.741,Z 237.912,A -85,B 0,C 180,E1 -14561.586,E2 -14561.586} C_VEL
LIN {X 0,Y 333.809,Z 237.906,A -85,B 0,C 180,E1 -14565.577,E2 -14565.577} C_VEL
LIN {X 0,Y 333.834,Z 237.894,A -85,B 0,C 180,E1 -14569.078,E2 -14569.078} C_VEL
LIN {X 0,Y 334.015,Z 237.87,A -85,B 0,C 180,E1 -14572.747,E2 -14572.747} C_VEL
LIN {X 0,Y 333.799,Z 237.904,A -85,B 0,C 180,E1 -14575.169,E2 -14575.169} C_VEL
LIN {X 0,Y 334.094,Z 237.86,A -85,B 0,C 180,E1 -14577.589,E2 -14577.589} C_VEL
LIN {X 0,Y 334.227,Z 237.851,A -85,B 0,C 180,E1 -14580,E2 -14580} C_VEL
LIN {X 0,Y 334.102,Z 237.86,A -85,B 0,C 180,E1 -14582.411,E2 -14582.411} C_VEL
LIN {X 0,Y 333.972,Z 237.879,A -85,B 0,C 180,E1 -14586.467,E2 -14586.467} C_VEL
LIN {X 0,Y 333.822,Z 237.901,A -85,B 0,C 180,E1 -14589.696,E2 -14589.696} C_VEL
LIN {X 0,Y 333.798,Z 237.898,A -85,B 0,C 180,E1 -14593.392,E2 -14593.392} C_VEL
LIN {X 0,Y 333.72,Z 237.911,A -85,B 0,C 180,E1 -14597.148,E2 -14597.148} C_VEL
LIN {X 0,Y 333.725,Z 237.914,A -85,B 0,C 180,E1 -14599.691,E2 -14599.691} C_VEL
LIN {X 0,Y 333.694,Z 237.907,A -85,B 0,C 180,E1 -14602.278,E2 -14602.278} C_VEL
LIN {X 0,Y 333.736,Z 237.904,A -85,B 0,C 180,E1 -14606.246,E2 -14606.246} C_VEL
LIN {X 0,Y 333.691,Z 237.919,A -85,B 0,C 180,E1 -14608.974,E2 -14608.974} C_VEL
LIN {X 0,Y 333.645,Z 237.923,A -85,B 0,C 180,E1 -14612.587,E2 -14612.587} C_VEL
LIN {X 0,Y 333.678,Z 237.915,A -85,B 0,C 180,E1 -14616.139,E2 -14616.139} C_VEL
LIN {X 0,Y 333.649,Z 237.922,A -85,B 0,C 180,E1 -14619.192,E2 -14619.192} C_VEL
LIN {X 0,Y 333.634,Z 237.926,A -85,B 0,C 180,E1 -14622.5,E2 -14622.5} C_VEL
LIN {X 0,Y 333.623,Z 237.923,A -85,B 0,C 180,E1 -14625.959,E2 -14625.959} C_VEL
LIN {X 0,Y 333.604,Z 237.932,A -85,B 0,C 180,E1 -14629.325,E2 -14629.325} C_VEL
LIN {X 0,Y 333.665,Z 237.929,A -85,B 0,C 180,E1 -14633.169,E2 -14633.169} C_VEL
LIN {X 0,Y 333.693,Z 237.956,A -85,B 0,C 180,E1 -14635.709,E2 -14635.709} C_VEL
LIN {X 0,Y 336.03,Z 248.098,A -85,B 0,C 180,E1 -14638.879,E2 -14638.879} C_VEL
LIN {X 0,Y 343.564,Z 265.939,A -85,B 0,C 180,E1 -14639.947,E2 -14639.947} C_VEL
LIN {X 0,Y 346.424,Z 278.453,A -85,B 0,C 180,E1 -14640.468,E2 -14640.468} C_VEL
LIN {X 0,Y 344.549,Z 355.851,A -85,B 0,C 180,E1 -14642.104,E2 -14642.104} C_VEL
LIN {X 0,Y 343.784,Z 369.817,A -85,B 0,C 180,E1 -14642.656,E2 -14642.656} C_VEL
LIN {X 0,Y 342.787,Z 382.787,A -85,B 0,C 180,E1 -14643.435,E2 -14643.435} C_VEL
LIN {X 0,Y 341.496,Z 394.595,A -85,B 0,C 180,E1 -14644.394,E2 -14644.394} C_VEL
LIN {X 0,Y 340.103,Z 405.957,A -85,B 0,C 180,E1 -14645.589,E2 -14645.589} C_VEL
LIN {X 0,Y 338.513,Z 416.129,A -85,B 0,C 180,E1 -14646.929,E2 -14646.929} C_VEL
LIN {X 0,Y 337.119,Z 426.113,A -85,B 0,C 180,E1 -14648.603,E2 -14648.603} C_VEL
LIN {X 0,Y 335.723,Z 434.857,A -85,B 0,C 180,E1 -14650.431,E2 -14650.431} C_VEL
LIN {X 0,Y 334.552,Z 441.798,A -85,B 0,C 180,E1 -14652.266,E2 -14652.266} C_VEL
LIN {X 0,Y 333.657,Z 447.334,A -85,B 0,C 180,E1 -14654.108,E2 -14654.108} C_VEL
LIN {X 0,Y 332.933,Z 452.109,A -85,B 0,C 180,E1 -14656.177,E2 -14656.177} C_VEL
LIN {X 0,Y 332.469,Z 454.895,A -85,B 0,C 180,E1 -14657.796,E2 -14657.796} C_VEL
LIN {X 0,Y 332.042,Z 457.695,A -85,B 0,C 180,E1 -14660.251,E2 -14660.251} C_VEL
LIN {X 0,Y 331.959,Z 458.447,A -85,B 0,C 180,E1 -14661.477,E2 -14661.477} C_VEL
LIN {X 0,Y 331.98,Z 458.799,A -85,B 0,C 180,E1 -14662.703,E2 -14662.703} C_VEL
LIN {X 0,Y 332.002,Z 458.721,A -85,B 0,C 180,E1 -14664.227,E2 -14664.227} C_VEL
LIN {X 0,Y 332.003,Z 457.521,A -85,B 0,C 180,E1 -14666.359,E2 -14666.359} C_VEL
LIN {X 0,Y 332.118,Z 454.642,A -85,B 0,C 180,E1 -14668.787,E2 -14668.787} C_VEL
LIN {X 0,Y 332.38,Z 451.353,A -85,B 0,C 180,E1 -14670.606,E2 -14670.606} C_VEL
LIN {X 0,Y 332.742,Z 447.008,A -85,B 0,C 180,E1 -14672.421,E2 -14672.421} C_VEL
LIN {X 0,Y 333.308,Z 441.481,A -85,B 0,C 180,E1 -14674.232,E2 -14674.232} C_VEL
LIN {X 0,Y 334.102,Z 434.586,A -85,B 0,C 180,E1 -14676.037,E2 -14676.037} C_VEL
LIN {X 0,Y 335.156,Z 425.943,A -85,B 0,C 180,E1 -14677.834,E2 -14677.834} C_VEL
LIN {X 0,Y 336.203,Z 417.099,A -85,B 0,C 180,E1 -14679.323,E2 -14679.323} C_VEL
LIN {X 0,Y 337.297,Z 407.383,A -85,B 0,C 180,E1 -14680.656,E2 -14680.656} C_VEL
LIN {X 0,Y 338.347,Z 396.715,A -85,B 0,C 180,E1 -14681.836,E2 -14681.836} C_VEL
LIN {X 0,Y 339.292,Z 384.768,A -85,B 0,C 180,E1 -14682.866,E2 -14682.866} C_VEL
LIN {X 0,Y 340.123,Z 372.167,A -85,B 0,C 180,E1 -14683.679,E2 -14683.679} C_VEL
LIN {X 0,Y 340.677,Z 358.969,A -85,B 0,C 180,E1 -14684.265,E2 -14684.265} C_VEL
LIN {X 0,Y 341.133,Z 341.614,A -85,B 0,C 180,E1 -14684.694,E2 -14684.694} C_VEL
LIN {X 0,Y 342.355,Z 276.029,A -85,B 0,C 180,E1 -14686.054,E2 -14686.054} C_VEL
LIN {X 0,Y 338.631,Z 255.85,A -85,B 0,C 180,E1 -14686.73,E2 -14686.73} C_VEL
LIN {X 0,Y 335.712,Z 247.628,A -85,B 0,C 180,E1 -14687.121,E2 -14687.121} C_VEL
LIN {X 0,Y 333.728,Z 237.916,A -85,B 0,C 180,E1 -14690.012,E2 -14690.012} C_VEL
LIN {X 0,Y 333.701,Z 237.919,A -85,B 0,C 180,E1 -14690.382,E2 -14690.382} C_VEL
LIN {X 0,Y 333.002,Z 238.004,A -85,B 0,C 180,E1 -14691.389,E2 -14691.389} C_VEL
LIN {X 0,Y 330.167,Z 238.358,A -85,B 0,C 180,E1 -14693.027,E2 -14693.027} C_VEL
LIN {X 0,Y 327.773,Z 238.657,A -85,B 0,C 180,E1 -14694.354,E2 -14694.354} C_VEL
LIN {X 0,Y 326.727,Z 238.785,A -85,B 0,C 180,E1 -14695.381,E2 -14695.381} C_VEL
LIN {X 0,Y 326.629,Z 238.795,A -85,B 0,C 180,E1 -14695.728,E2 -14695.728} C_VEL
LIN {X 0,Y 326.626,Z 238.796,A -85,B 0,C 180,E1 -14699.662,E2 -14699.662} C_VEL
LIN {X 0,Y 326.619,Z 238.8,A -85,B 0,C 180,E1 -14702.946,E2 -14702.946} C_VEL
LIN {X 0,Y 326.614,Z 238.797,A -85,B 0,C 180,E1 -14705.519,E2 -14705.519} C_VEL
LIN {X 0,Y 326.613,Z 238.799,A -85,B 0,C 180,E1 -14709.227,E2 -14709.227} C_VEL
LIN {X 0,Y 326.584,Z 238.804,A -85,B 0,C 180,E1 -14712.973,E2 -14712.973} C_VEL
LIN {X 0,Y 326.582,Z 238.804,A -85,B 0,C 180,E1 -14717.027,E2 -14717.027} C_VEL
LIN {X 0,Y 326.612,Z 238.802,A -85,B 0,C 180,E1 -14720.773,E2 -14720.773} C_VEL
LIN {X 0,Y 326.614,Z 238.802,A -85,B 0,C 180,E1 -14724.48,E2 -14724.48} C_VEL
LIN {X 0,Y 326.609,Z 238.794,A -85,B 0,C 180,E1 -14727.455,E2 -14727.455} C_VEL
LIN {X 0,Y 326.649,Z 238.794,A -85,B 0,C 180,E1 -14730.339,E2 -14730.339} C_VEL
LIN {X 0,Y 326.691,Z 238.792,A -85,B 0,C 180,E1 -14734.516,E2 -14734.516} C_VEL
LIN {X 0,Y 326.649,Z 238.792,A -85,B 0,C 180,E1 -14738.545,E2 -14738.545} C_VEL
LIN {X 0,Y 326.745,Z 238.781,A -85,B 0,C 180,E1 -14741.177,E2 -14741.177} C_VEL
LIN {X 0,Y 326.764,Z 238.777,A -85,B 0,C 180,E1 -14745.433,E2 -14745.433} C_VEL
LIN {X 0,Y 326.759,Z 238.777,A -85,B 0,C 180,E1 -14748.838,E2 -14748.838} C_VEL
LIN {X 0,Y 326.919,Z 238.763,A -85,B 0,C 180,E1 -14752.589,E2 -14752.589} C_VEL
LIN {X 0,Y 326.769,Z 238.779,A -85,B 0,C 180,E1 -14755.065,E2 -14755.065} C_VEL
LIN {X 0,Y 327.046,Z 238.742,A -85,B 0,C 180,E1 -14757.537,E2 -14757.537} C_VEL
LIN {X 0,Y 327.178,Z 238.727,A -85,B 0,C 180,E1 -14760,E2 -14760} C_VEL
LIN {X 0,Y 327.043,Z 238.748,A -85,B 0,C 180,E1 -14762.463,E2 -14762.463} C_VEL
LIN {X 0,Y 326.996,Z 238.751,A -85,B 0,C 180,E1 -14766.169,E2 -14766.169} C_VEL
LIN {X 0,Y 326.915,Z 238.764,A -85,B 0,C 180,E1 -14768.655,E2 -14768.655} C_VEL
LIN {X 0,Y 326.735,Z 238.784,A -85,B 0,C 180,E1 -14772.421,E2 -14772.421} C_VEL
LIN {X 0,Y 326.751,Z 238.783,A -85,B 0,C 180,E1 -14774.958,E2 -14774.958} C_VEL
LIN {X 0,Y 326.662,Z 238.794,A -85,B 0,C 180,E1 -14778.827,E2 -14778.827} C_VEL
LIN {X 0,Y 326.601,Z 238.802,A -85,B 0,C 180,E1 -14782.789,E2 -14782.789} C_VEL
LIN {X 0,Y 326.639,Z 238.793,A -85,B 0,C 180,E1 -14785.488,E2 -14785.488} C_VEL
LIN {X 0,Y 326.622,Z 238.799,A -85,B 0,C 180,E1 -14788.254,E2 -14788.254} C_VEL
LIN {X 0,Y 326.573,Z 238.803,A -85,B 0,C 180,E1 -14791.097,E2 -14791.097} C_VEL
LIN {X 0,Y 326.607,Z 238.799,A -85,B 0,C 180,E1 -14794.019,E2 -14794.019} C_VEL
LIN {X 0,Y 326.623,Z 238.797,A -85,B 0,C 180,E1 -14797.238,E2 -14797.238} C_VEL
LIN {X 0,Y 326.544,Z 238.807,A -85,B 0,C 180,E1 -14801.125,E2 -14801.125} C_VEL
LIN {X 0,Y 326.561,Z 238.804,A -85,B 0,C 180,E1 -14803.526,E2 -14803.526} C_VEL
LIN {X 0,Y 326.575,Z 238.803,A -85,B 0,C 180,E1 -14807.028,E2 -14807.028} C_VEL
LIN {X 0,Y 326.611,Z 238.801,A -85,B 0,C 180,E1 -14810.773,E2 -14810.773} C_VEL
LIN {X 0,Y 326.614,Z 238.803,A -85,B 0,C 180,E1 -14814.481,E2 -14814.481} C_VEL
LIN {X 0,Y 326.609,Z 238.8,A -85,B 0,C 180,E1 -14817.456,E2 -14817.456} C_VEL
LIN {X 0,Y 326.64,Z 238.832,A -85,B 0,C 180,E1 -14819.506,E2 -14819.506} C_VEL
LIN {X 0,Y 329.218,Z 251.154,A -85,B 0,C 180,E1 -14823.023,E2 -14823.023} C_VEL
LIN {X 0,Y 330.315,Z 257.702,A -85,B 0,C 180,E1 -14824.816,E2 -14824.816} C_VEL
LIN {X 0,Y 329.657,Z 264.414,A -85,B 0,C 180,E1 -14826.513,E2 -14826.513} C_VEL
LIN {X 0,Y 334.115,Z 293.751,A -85,B 0,C 180,E1 -14827.479,E2 -14827.479} C_VEL
LIN {X 0,Y 335.265,Z 303.145,A -85,B 0,C 180,E1 -14827.76,E2 -14827.76} C_VEL
LIN {X 0,Y 333.892,Z 373.227,A -85,B 0,C 180,E1 -14829.275,E2 -14829.275} C_VEL
LIN {X 0,Y 333.117,Z 387.142,A -85,B 0,C 180,E1 -14829.83,E2 -14829.83} C_VEL
LIN {X 0,Y 332.13,Z 400.103,A -85,B 0,C 180,E1 -14830.613,E2 -14830.613} C_VEL
LIN {X 0,Y 331.046,Z 411.908,A -85,B 0,C 180,E1 -14831.591,E2 -14831.591} C_VEL
LIN {X 0,Y 329.82,Z 423.284,A -85,B 0,C 180,E1 -14832.803,E2 -14832.803} C_VEL
LIN {X 0,Y 328.66,Z 433.735,A -85,B 0,C 180,E1 -14834.212,E2 -14834.212} C_VEL
LIN {X 0,Y 327.674,Z 442.742,A -85,B 0,C 180,E1 -14835.72,E2 -14835.72} C_VEL
LIN {X 0,Y 326.648,Z 451.708,A -85,B 0,C 180,E1 -14837.575,E2 -14837.575} C_VEL
LIN {X 0,Y 325.877,Z 458.909,A -85,B 0,C 180,E1 -14839.437,E2 -14839.437} C_VEL
LIN {X 0,Y 325.367,Z 464.643,A -85,B 0,C 180,E1 -14841.303,E2 -14841.303} C_VEL
LIN {X 0,Y 325.052,Z 469.153,A -85,B 0,C 180,E1 -14843.17,E2 -14843.17} C_VEL
LIN {X 0,Y 324.897,Z 472.572,A -85,B 0,C 180,E1 -14845.036,E2 -14845.036} C_VEL
LIN {X 0,Y 324.9,Z 474.27,A -85,B 0,C 180,E1 -14846.279,E2 -14846.279} C_VEL
LIN {X 0,Y 324.838,Z 475.558,A -85,B 0,C 180,E1 -14847.52,E2 -14847.52} C_VEL
LIN {X 0,Y 324.833,Z 476.452,A -85,B 0,C 180,E1 -14848.76,E2 -14848.76} C_VEL
LIN {X 0,Y 324.874,Z 476.922,A -85,B 0,C 180,E1 -14850,E2 -14850} C_VEL
LIN {X 0,Y 324.833,Z 476.649,A -85,B 0,C 180,E1 -14852.48,E2 -14852.48} C_VEL
LIN {X 0,Y 324.875,Z 475.937,A -85,B 0,C 180,E1 -14853.721,E2 -14853.721} C_VEL
LIN {X 0,Y 324.982,Z 473.757,A -85,B 0,C 180,E1 -14855.851,E2 -14855.851} C_VEL
LIN {X 0,Y 325.297,Z 470.124,A -85,B 0,C 180,E1 -14858.073,E2 -14858.073} C_VEL
LIN {X 0,Y 325.855,Z 465.954,A -85,B 0,C 180,E1 -14859.936,E2 -14859.936} C_VEL
LIN {X 0,Y 326.759,Z 459.615,A -85,B 0,C 180,E1 -14862.105,E2 -14862.105} C_VEL
LIN {X 0,Y 328.001,Z 452.727,A -85,B 0,C 180,E1 -14863.949,E2 -14863.949} C_VEL
LIN {X 0,Y 329.39,Z 444.125,A -85,B 0,C 180,E1 -14865.786,E2 -14865.786} C_VEL
LIN {X 0,Y 330.731,Z 435.321,A -85,B 0,C 180,E1 -14867.307,E2 -14867.307} C_VEL
LIN {X 0,Y 332.441,Z 424.5,A -85,B 0,C 180,E1 -14868.808,E2 -14868.808} C_VEL
LIN {X 0,Y 333.96,Z 413.615,A -85,B 0,C 180,E1 -14869.997,E2 -14869.997} C_VEL
LIN {X 0,Y 335.504,Z 401.422,A -85,B 0,C 180,E1 -14871.022,E2 -14871.022} C_VEL
LIN {X 0,Y 336.751,Z 388.629,A -85,B 0,C 180,E1 -14871.823,E2 -14871.823} C_VEL
LIN {X 0,Y 337.633,Z 375.802,A -85,B 0,C 180,E1 -14872.365,E2 -14872.365} C_VEL
LIN {X 0,Y 338.297,Z 357.755,A -85,B 0,C 180,E1 -14872.801,E2 -14872.801} C_VEL
LIN {X 0,Y 339.375,Z 303.299,A -85,B 0,C 180,E1 -14873.969,E2 -14873.969} C_VEL
LIN {X 0,Y 335.092,Z 279.366,A -85,B 0,C 180,E1 -14874.892,E2 -14874.892} C_VEL
LIN {X 0,Y 331.835,Z 264.145,A -85,B 0,C 180,E1 -14875.556,E2 -14875.556} C_VEL
LIN {X 0,Y 331.194,Z 259.127,A -85,B 0,C 180,E1 -14876.969,E2 -14876.969} C_VEL
LIN {X 0,Y 329.246,Z 249.738,A -85,B 0,C 180,E1 -14879.755,E2 -14879.755} C_VEL
LIN {X 0,Y 326.613,Z 238.798,A -85,B 0,C 180,E1 -14883.2,E2 -14883.2} C_VEL
LIN {X 0,Y 326.631,Z 238.8,A -85,B 0,C 180,E1 -14887.047,E2 -14887.047} C_VEL
LIN {X 0,Y 326.592,Z 238.804,A -85,B 0,C 180,E1 -14890.209,E2 -14890.209} C_VEL
LIN {X 0,Y 326.562,Z 238.809,A -85,B 0,C 180,E1 -14893.526,E2 -14893.526} C_VEL
LIN {X 0,Y 326.574,Z 238.807,A -85,B 0,C 180,E1 -14897.029,E2 -14897.029} C_VEL
LIN {X 0,Y 326.582,Z 238.806,A -85,B 0,C 180,E1 -14901.386,E2 -14901.386} C_VEL
LIN {X 0,Y 326.619,Z 238.798,A -85,B 0,C 180,E1 -14904.851,E2 -14904.851} C_VEL
LIN {X 0,Y 326.608,Z 238.797,A -85,B 0,C 180,E1 -14907.456,E2 -14907.456} C_VEL
LIN {X 0,Y 326.625,Z 238.789,A -85,B 0,C 180,E1 -14910.337,E2 -14910.337} C_VEL
LIN {X 0,Y 326.628,Z 238.8,A -85,B 0,C 180,E1 -14913.137,E2 -14913.137} C_VEL
LIN {X 0,Y 326.644,Z 238.797,A -85,B 0,C 180,E1 -14915.871,E2 -14915.871} C_VEL
LIN {X 0,Y 326.631,Z 238.797,A -85,B 0,C 180,E1 -14919.863,E2 -14919.863} C_VEL
LIN {X 0,Y 326.665,Z 238.789,A -85,B 0,C 180,E1 -14922.47,E2 -14922.47} C_VEL
LIN {X 0,Y 326.76,Z 238.779,A -85,B 0,C 180,E1 -14926.315,E2 -14926.315} C_VEL
LIN {X 0,Y 326.813,Z 238.774,A -85,B 0,C 180,E1 -14930.094,E2 -14930.094} C_VEL
LIN {X 0,Y 326.968,Z 238.748,A -85,B 0,C 180,E1 -14932.59,E2 -14932.59} C_VEL
LIN {X 0,Y 326.991,Z 238.748,A -85,B 0,C 180,E1 -14933.831,E2 -14933.831} C_VEL
LIN {X 0,Y 327.035,Z 238.739,A -85,B 0,C 180,E1 -14937.537,E2 -14937.537} C_VEL
LIN {X 0,Y 327.178,Z 238.729,A -85,B 0,C 180,E1 -14940,E2 -14940} C_VEL
LIN {X 0,Y 327.043,Z 238.739,A -85,B 0,C 180,E1 -14942.463,E2 -14942.463} C_VEL
LIN {X 0,Y 326.933,Z 238.756,A -85,B 0,C 180,E1 -14946.455,E2 -14946.455} C_VEL
LIN {X 0,Y 326.784,Z 238.779,A -85,B 0,C 180,E1 -14949.907,E2 -14949.907} C_VEL
LIN {X 0,Y 326.76,Z 238.774,A -85,B 0,C 180,E1 -14953.686,E2 -14953.686} C_VEL
LIN {X 0,Y 326.665,Z 238.786,A -85,B 0,C 180,E1 -14957.53,E2 -14957.53} C_VEL
LIN {X 0,Y 326.659,Z 238.792,A -85,B 0,C 180,E1 -14960.135,E2 -14960.135} C_VEL
LIN {X 0,Y 326.653,Z 238.793,A -85,B 0,C 180,E1 -14964.129,E2 -14964.129} C_VEL
LIN {X 0,Y 326.684,Z 238.783,A -85,B 0,C 180,E1 -14966.858,E2 -14966.858} C_VEL
LIN {X 0,Y 326.635,Z 238.792,A -85,B 0,C 180,E1 -14970.61,E2 -14970.61} C_VEL
LIN {X 0,Y 326.608,Z 238.8,A -85,B 0,C 180,E1 -14974.02,E2 -14974.02} C_VEL
LIN {X 0,Y 326.63,Z 238.797,A -85,B 0,C 180,E1 -14977.239,E2 -14977.239} C_VEL
LIN {X 0,Y 326.579,Z 238.805,A -85,B 0,C 180,E1 -14981.131,E2 -14981.131} C_VEL
LIN {X 0,Y 326.557,Z 238.809,A -85,B 0,C 180,E1 -14984.748,E2 -14984.748} C_VEL
LIN {X 0,Y 326.565,Z 238.812,A -85,B 0,C 180,E1 -14988.152,E2 -14988.152} C_VEL
LIN {X 0,Y 326.584,Z 238.81,A -85,B 0,C 180,E1 -14991.386,E2 -14991.386} C_VEL
LIN {X 0,Y 326.665,Z 238.81,A -85,B 0,C 180,E1 -14995.171,E2 -14995.171} C_VEL
LIN {X 0,Y 328.851,Z 248.226,A -85,B 0,C 180,E1 -14998.221,E2 -14998.221} C_VEL
LIN {X 0,Y 337.346,Z 268.084,A -85,B 0,C 180,E1 -14999.466,E2 -14999.466} C_VEL
LIN {X 0,Y 340.069,Z 280.16,A -85,B 0,C 180,E1 -14999.981,E2 -14999.981} C_VEL
LIN {X 0,Y 338.104,Z 356.013,A -85,B 0,C 180,E1 -15001.609,E2 -15001.609} C_VEL
LIN {X 0,Y 337.314,Z 369.991,A -85,B 0,C 180,E1 -15002.171,E2 -15002.171} C_VEL
LIN {X 0,Y 336.267,Z 382.967,A -85,B 0,C 180,E1 -15002.962,E2 -15002.962} C_VEL
LIN {X 0,Y 335.018,Z 393.977,A -85,B 0,C 180,E1 -15003.862,E2 -15003.862} C_VEL
LIN {X 0,Y 333.528,Z 405.486,A -85,B 0,C 180,E1 -15005.075,E2 -15005.075} C_VEL
LIN {X 0,Y 331.952,Z 415.82,A -85,B 0,C 180,E1 -15006.446,E2 -15006.446} C_VEL
LIN {X 0,Y 330.665,Z 424.249,A -85,B 0,C 180,E1 -15007.836,E2 -15007.836} C_VEL
LIN {X 0,Y 329.121,Z 433.358,A -85,B 0,C 180,E1 -15009.696,E2 -15009.696} C_VEL
LIN {X 0,Y 327.891,Z 440.675,A -85,B 0,C 180,E1 -15011.57,E2 -15011.57} C_VEL
LIN {X 0,Y 326.999,Z 445.601,A -85,B 0,C 180,E1 -15013.133,E2 -15013.133} C_VEL
LIN {X 0,Y 326.213,Z 450.366,A -85,B 0,C 180,E1 -15015.017,E2 -15015.017} C_VEL
LIN {X 0,Y 325.635,Z 453.999,A -85,B 0,C 180,E1 -15016.902,E2 -15016.902} C_VEL
LIN {X 0,Y 325.156,Z 456.602,A -85,B 0,C 180,E1 -15018.783,E2 -15018.783} C_VEL
LIN {X 0,Y 324.963,Z 457.822,A -85,B 0,C 180,E1 -15020.037,E2 -15020.037} C_VEL
LIN {X 0,Y 324.896,Z 458.613,A -85,B 0,C 180,E1 -15021.291,E2 -15021.291} C_VEL
LIN {X 0,Y 324.943,Z 458.976,A -85,B 0,C 180,E1 -15023.792,E2 -15023.792} C_VEL
LIN {X 0,Y 324.881,Z 458.589,A -85,B 0,C 180,E1 -15025.036,E2 -15025.036} C_VEL
LIN {X 0,Y 324.928,Z 457.789,A -85,B 0,C 180,E1 -15026.28,E2 -15026.28} C_VEL
LIN {X 0,Y 325.015,Z 454.953,A -85,B 0,C 180,E1 -15028.761,E2 -15028.761} C_VEL
LIN {X 0,Y 325.309,Z 451.707,A -85,B 0,C 180,E1 -15030.619,E2 -15030.619} C_VEL
LIN {X 0,Y 325.681,Z 447.409,A -85,B 0,C 180,E1 -15032.474,E2 -15032.474} C_VEL
LIN {X 0,Y 326.255,Z 441.934,A -85,B 0,C 180,E1 -15034.324,E2 -15034.324} C_VEL
LIN {X 0,Y 327.082,Z 435.102,A -85,B 0,C 180,E1 -15036.167,E2 -15036.167} C_VEL
LIN {X 0,Y 328.169,Z 426.552,A -85,B 0,C 180,E1 -15038.002,E2 -15038.002} C_VEL
LIN {X 0,Y 329.236,Z 417.79,A -85,B 0,C 180,E1 -15039.522,E2 -15039.522} C_VEL
LIN {X 0,Y 330.499,Z 407.007,A -85,B 0,C 180,E1 -15041.033,E2 -15041.033} C_VEL
LIN {X 0,Y 331.55,Z 396.151,A -85,B 0,C 180,E1 -15042.238,E2 -15042.238} C_VEL
LIN {X 0,Y 332.584,Z 383.995,A -85,B 0,C 180,E1 -15043.286,E2 -15043.286} C_VEL
LIN {X 0,Y 333.341,Z 372.978,A -85,B 0,C 180,E1 -15044.004,E2 -15044.004} C_VEL
LIN {X 0,Y 333.909,Z 360.358,A -85,B 0,C 180,E1 -15044.597,E2 -15044.597} C_VEL
LIN {X 0,Y 334.305,Z 347.185,A -85,B 0,C 180,E1 -15044.962,E2 -15044.962} C_VEL
LIN {X 0,Y 335.692,Z 276.802,A -85,B 0,C 180,E1 -15046.449,E2 -15046.449} C_VEL
LIN {X 0,Y 332.248,Z 258.269,A -85,B 0,C 180,E1 -15047.088,E2 -15047.088} C_VEL
LIN {X 0,Y 328.556,Z 247.857,A -85,B 0,C 180,E1 -15047.586,E2 -15047.586} C_VEL
LIN {X 0,Y 326.671,Z 238.795,A -85,B 0,C 180,E1 -15050.34,E2 -15050.34} C_VEL
LIN {X 0,Y 326.645,Z 238.796,A -85,B 0,C 180,E1 -15054.129,E2 -15054.129} C_VEL
LIN {X 0,Y 326.629,Z 238.795,A -85,B 0,C 180,E1 -15055.728,E2 -15055.728} C_VEL
LIN {X 0,Y 325.934,Z 238.888,A -85,B 0,C 180,E1 -15056.757,E2 -15056.757} C_VEL
LIN {X 0,Y 323.088,Z 239.241,A -85,B 0,C 180,E1 -15058.432,E2 -15058.432} C_VEL
LIN {X 0,Y 320.682,Z 239.542,A -85,B 0,C 180,E1 -15059.788,E2 -15059.788} C_VEL
LIN {X 0,Y 319.632,Z 239.672,A -85,B 0,C 180,E1 -15060.838,E2 -15060.838} C_VEL
LIN {X 0,Y 319.537,Z 239.681,A -85,B 0,C 180,E1 -15061.193,E2 -15061.193} C_VEL
LIN {X 0,Y 319.562,Z 239.68,A -85,B 0,C 180,E1 -15064.876,E2 -15064.876} C_VEL
LIN {X 0,Y 319.559,Z 239.677,A -85,B 0,C 180,E1 -15068.01,E2 -15068.01} C_VEL
LIN {X 0,Y 319.527,Z 239.68,A -85,B 0,C 180,E1 -15071.597,E2 -15071.597} C_VEL
LIN {X 0,Y 319.517,Z 239.687,A -85,B 0,C 180,E1 -15074.738,E2 -15074.738} C_VEL
LIN {X 0,Y 319.526,Z 239.684,A -85,B 0,C 180,E1 -15078.403,E2 -15078.403} C_VEL
LIN {X 0,Y 319.544,Z 239.678,A -85,B 0,C 180,E1 -15081.988,E2 -15081.988} C_VEL
LIN {X 0,Y 319.561,Z 239.676,A -85,B 0,C 180,E1 -15085.123,E2 -15085.123} C_VEL
LIN {X 0,Y 319.567,Z 239.675,A -85,B 0,C 180,E1 -15089.059,E2 -15089.059} C_VEL
LIN {X 0,Y 319.607,Z 239.674,A -85,B 0,C 180,E1 -15092.498,E2 -15092.498} C_VEL
LIN {X 0,Y 319.605,Z 239.668,A -85,B 0,C 180,E1 -15095.304,E2 -15095.304} C_VEL
LIN {X 0,Y 319.599,Z 239.665,A -85,B 0,C 180,E1 -15098.048,E2 -15098.048} C_VEL
LIN {X 0,Y 319.69,Z 239.661,A -85,B 0,C 180,E1 -15100.962,E2 -15100.962} C_VEL
LIN {X 0,Y 319.732,Z 239.653,A -85,B 0,C 180,E1 -15105.276,E2 -15105.276} C_VEL
LIN {X 0,Y 319.716,Z 239.653,A -85,B 0,C 180,E1 -15108.589,E2 -15108.589} C_VEL
LIN {X 0,Y 319.857,Z 239.64,A -85,B 0,C 180,E1 -15112.424,E2 -15112.424} C_VEL
LIN {X 0,Y 319.737,Z 239.656,A -85,B 0,C 180,E1 -15114.956,E2 -15114.956} C_VEL
LIN {X 0,Y 319.989,Z 239.62,A -85,B 0,C 180,E1 -15117.482,E2 -15117.482} C_VEL
LIN {X 0,Y 320.131,Z 239.605,A -85,B 0,C 180,E1 -15120,E2 -15120} C_VEL
LIN {X 0,Y 319.986,Z 239.628,A -85,B 0,C 180,E1 -15122.518,E2 -15122.518} C_VEL
LIN {X 0,Y 319.952,Z 239.63,A -85,B 0,C 180,E1 -15126.305,E2 -15126.305} C_VEL
LIN {X 0,Y 319.843,Z 239.643,A -85,B 0,C 180,E1 -15128.848,E2 -15128.848} C_VEL
LIN {X 0,Y 319.683,Z 239.665,A -85,B 0,C 180,E1 -15132.7,E2 -15132.7} C_VEL
LIN {X 0,Y 319.679,Z 239.662,A -85,B 0,C 180,E1 -15135.296,E2 -15135.296} C_VEL
LIN {X 0,Y 319.588,Z 239.672,A -85,B 0,C 180,E1 -15139.26,E2 -15139.26} C_VEL
LIN {X 0,Y 319.557,Z 239.676,A -85,B 0,C 180,E1 -15143.32,E2 -15143.32} C_VEL
LIN {X 0,Y 319.574,Z 239.674,A -85,B 0,C 180,E1 -15146.093,E2 -15146.093} C_VEL
LIN {X 0,Y 319.552,Z 239.679,A -85,B 0,C 180,E1 -15148.937,E2 -15148.937} C_VEL
LIN {X 0,Y 319.524,Z 239.681,A -85,B 0,C 180,E1 -15151.863,E2 -15151.863} C_VEL
LIN {X 0,Y 319.579,Z 239.673,A -85,B 0,C 180,E1 -15155.543,E2 -15155.543} C_VEL
LIN {X 0,Y 319.528,Z 239.68,A -85,B 0,C 180,E1 -15159.662,E2 -15159.662} C_VEL
LIN {X 0,Y 319.52,Z 239.681,A -85,B 0,C 180,E1 -15163.46,E2 -15163.46} C_VEL
LIN {X 0,Y 319.553,Z 239.678,A -85,B 0,C 180,E1 -15167.016,E2 -15167.016} C_VEL
LIN {X 0,Y 319.547,Z 239.681,A -85,B 0,C 180,E1 -15170.371,E2 -15170.371} C_VEL
LIN {X 0,Y 319.56,Z 239.677,A -85,B 0,C 180,E1 -15173.573,E2 -15173.573} C_VEL
LIN {X 0,Y 319.578,Z 239.68,A -85,B 0,C 180,E1 -15176.687,E2 -15176.687} C_VEL
LIN {X 0,Y 319.584,Z 239.75,A -85,B 0,C 180,E1 -15179.148,E2 -15179.148} C_VEL
LIN {X 0,Y 321.949,Z 250.69,A -85,B 0,C 180,E1 -15182.362,E2 -15182.362} C_VEL
LIN {X 0,Y 323.304,Z 258.556,A -85,B 0,C 180,E1 -15184.575,E2 -15184.575} C_VEL
LIN {X 0,Y 322.83,Z 264.214,A -85,B 0,C 180,E1 -15186.045,E2 -15186.045} C_VEL
LIN {X 0,Y 327.08,Z 291.863,A -85,B 0,C 180,E1 -15186.988,E2 -15186.988} C_VEL
LIN {X 0,Y 328.581,Z 303.731,A -85,B 0,C 180,E1 -15187.356,E2 -15187.356} C_VEL
LIN {X 0,Y 327.172,Z 372.655,A -85,B 0,C 180,E1 -15188.87,E2 -15188.87} C_VEL
LIN {X 0,Y 326.438,Z 385.931,A -85,B 0,C 180,E1 -15189.398,E2 -15189.398} C_VEL
LIN {X 0,Y 325.523,Z 398.112,A -85,B 0,C 180,E1 -15190.121,E2 -15190.121} C_VEL
LIN {X 0,Y 324.485,Z 409.585,A -85,B 0,C 180,E1 -15191.042,E2 -15191.042} C_VEL
LIN {X 0,Y 323.166,Z 421.357,A -85,B 0,C 180,E1 -15192.274,E2 -15192.274} C_VEL
LIN {X 0,Y 321.889,Z 432.138,A -85,B 0,C 180,E1 -15193.706,E2 -15193.706} C_VEL
LIN {X 0,Y 321.011,Z 440.571,A -85,B 0,C 180,E1 -15195.093,E2 -15195.093} C_VEL
LIN {X 0,Y 320.036,Z 448.525,A -85,B 0,C 180,E1 -15196.669,E2 -15196.669} C_VEL
LIN {X 0,Y 319.034,Z 456.28,A -85,B 0,C 180,E1 -15198.565,E2 -15198.565} C_VEL
LIN {X 0,Y 318.469,Z 462.508,A -85,B 0,C 180,E1 -15200.473,E2 -15200.473} C_VEL
LIN {X 0,Y 318.067,Z 467.446,A -85,B 0,C 180,E1 -15202.382,E2 -15202.382} C_VEL
LIN {X 0,Y 317.874,Z 471.137,A -85,B 0,C 180,E1 -15204.226,E2 -15204.226} C_VEL
LIN {X 0,Y 317.808,Z 474.014,A -85,B 0,C 180,E1 -15206.196,E2 -15206.196} C_VEL
LIN {X 0,Y 317.76,Z 475.316,A -85,B 0,C 180,E1 -15207.465,E2 -15207.465} C_VEL
LIN {X 0,Y 317.744,Z 476.223,A -85,B 0,C 180,E1 -15208.733,E2 -15208.733} C_VEL
LIN {X 0,Y 317.781,Z 476.719,A -85,B 0,C 180,E1 -15210,E2 -15210} C_VEL
LIN {X 0,Y 317.754,Z 476.472,A -85,B 0,C 180,E1 -15212.535,E2 -15212.535} C_VEL
LIN {X 0,Y 317.785,Z 475.773,A -85,B 0,C 180,E1 -15213.804,E2 -15213.804} C_VEL
LIN {X 0,Y 317.88,Z 473.853,A -85,B 0,C 180,E1 -15215.786,E2 -15215.786} C_VEL
LIN {X 0,Y 318.244,Z 470.029,A -85,B 0,C 180,E1 -15218.253,E2 -15218.253} C_VEL
LIN {X 0,Y 318.85,Z 465.89,A -85,B 0,C 180,E1 -15220.156,E2 -15220.156} C_VEL
LIN {X 0,Y 319.8,Z 459.584,A -85,B 0,C 180,E1 -15222.373,E2 -15222.373} C_VEL
LIN {X 0,Y 321.097,Z 452.733,A -85,B 0,C 180,E1 -15224.255,E2 -15224.255} C_VEL
LIN {X 0,Y 322.55,Z 444.197,A -85,B 0,C 180,E1 -15226.129,E2 -15226.129} C_VEL
LIN {X 0,Y 323.954,Z 435.448,A -85,B 0,C 180,E1 -15227.681,E2 -15227.681} C_VEL
LIN {X 0,Y 325.728,Z 424.694,A -85,B 0,C 180,E1 -15229.21,E2 -15229.21} C_VEL
LIN {X 0,Y 327.321,Z 413.945,A -85,B 0,C 180,E1 -15230.421,E2 -15230.421} C_VEL
LIN {X 0,Y 328.919,Z 401.888,A -85,B 0,C 180,E1 -15231.464,E2 -15231.464} C_VEL
LIN {X 0,Y 330.191,Z 389.317,A -85,B 0,C 180,E1 -15232.28,E2 -15232.28} C_VEL
LIN {X 0,Y 331.12,Z 377.079,A -85,B 0,C 180,E1 -15232.831,E2 -15232.831} C_VEL
LIN {X 0,Y 331.706,Z 363.346,A -85,B 0,C 180,E1 -15233.201,E2 -15233.201} C_VEL
LIN {X 0,Y 333.016,Z 304.117,A -85,B 0,C 180,E1 -15234.488,E2 -15234.488} C_VEL
LIN {X 0,Y 328.288,Z 278.068,A -85,B 0,C 180,E1 -15235.534,E2 -15235.534} C_VEL
LIN {X 0,Y 325.309,Z 265.413,A -85,B 0,C 180,E1 -15236.121,E2 -15236.121} C_VEL
LIN {X 0,Y 324.867,Z 263.735,A -85,B 0,C 180,E1 -15236.263,E2 -15236.263} C_VEL
LIN {X 0,Y 322.647,Z 252.492,A -85,B 0,C 180,E1 -15239.639,E2 -15239.639} C_VEL
LIN {X 0,Y 319.892,Z 241.034,A -85,B 0,C 180,E1 -15243.315,E2 -15243.315} C_VEL
LIN {X 0,Y 319.577,Z 239.677,A -85,B 0,C 180,E1 -15243.825,E2 -15243.825} C_VEL
LIN {X 0,Y 319.555,Z 239.681,A -85,B 0,C 180,E1 -15247.65,E2 -15247.65} C_VEL
LIN {X 0,Y 319.529,Z 239.685,A -85,B 0,C 180,E1 -15251.288,E2 -15251.288} C_VEL
LIN {X 0,Y 319.488,Z 239.688,A -85,B 0,C 180,E1 -15254.743,E2 -15254.743} C_VEL
LIN {X 0,Y 319.553,Z 239.681,A -85,B 0,C 180,E1 -15257.016,E2 -15257.016} C_VEL
LIN {X 0,Y 319.545,Z 239.679,A -85,B 0,C 180,E1 -15260.371,E2 -15260.371} C_VEL
LIN {X 0,Y 319.58,Z 239.674,A -85,B 0,C 180,E1 -15264.457,E2 -15264.457} C_VEL
LIN {X 0,Y 319.525,Z 239.682,A -85,B 0,C 180,E1 -15268.137,E2 -15268.137} C_VEL
LIN {X 0,Y 319.594,Z 239.672,A -85,B 0,C 180,E1 -15271.596,E2 -15271.596} C_VEL
LIN {X 0,Y 319.583,Z 239.67,A -85,B 0,C 180,E1 -15275.302,E2 -15275.302} C_VEL
LIN {X 0,Y 319.568,Z 239.672,A -85,B 0,C 180,E1 -15278.046,E2 -15278.046} C_VEL
LIN {X 0,Y 319.625,Z 239.667,A -85,B 0,C 180,E1 -15282.071,E2 -15282.071} C_VEL
LIN {X 0,Y 319.733,Z 239.656,A -85,B 0,C 180,E1 -15286.008,E2 -15286.008} C_VEL
LIN {X 0,Y 319.758,Z 239.654,A -85,B 0,C 180,E1 -15289.873,E2 -15289.873} C_VEL
LIN {X 0,Y 319.927,Z 239.624,A -85,B 0,C 180,E1 -15292.426,E2 -15292.426} C_VEL
LIN {X 0,Y 319.738,Z 239.654,A -85,B 0,C 180,E1 -15294.956,E2 -15294.956} C_VEL
LIN {X 0,Y 319.978,Z 239.618,A -85,B 0,C 180,E1 -15297.482,E2 -15297.482} C_VEL
LIN {X 0,Y 320.131,Z 239.606,A -85,B 0,C 180,E1 -15300,E2 -15300} C_VEL
LIN {X 0,Y 319.987,Z 239.618,A -85,B 0,C 180,E1 -15302.518,E2 -15302.518} C_VEL
LIN {X 0,Y 319.898,Z 239.633,A -85,B 0,C 180,E1 -15306.435,E2 -15306.435} C_VEL
LIN {X 0,Y 319.737,Z 239.656,A -85,B 0,C 180,E1 -15310.128,E2 -15310.128} C_VEL
LIN {X 0,Y 319.733,Z 239.651,A -85,B 0,C 180,E1 -15313.992,E2 -15313.992} C_VEL
LIN {X 0,Y 319.625,Z 239.66,A -85,B 0,C 180,E1 -15317.929,E2 -15317.929} C_VEL
LIN {X 0,Y 319.613,Z 239.669,A -85,B 0,C 180,E1 -15320.599,E2 -15320.599} C_VEL
LIN {X 0,Y 319.572,Z 239.671,A -85,B 0,C 180,E1 -15323.32,E2 -15323.32} C_VEL
LIN {X 0,Y 319.619,Z 239.663,A -85,B 0,C 180,E1 -15326.09,E2 -15326.09} C_VEL
LIN {X 0,Y 319.582,Z 239.676,A -85,B 0,C 180,E1 -15328.935,E2 -15328.935} C_VEL
LIN {X 0,Y 319.532,Z 239.683,A -85,B 0,C 180,E1 -15331.862,E2 -15331.862} C_VEL
LIN {X 0,Y 319.582,Z 239.675,A -85,B 0,C 180,E1 -15335.543,E2 -15335.543} C_VEL
LIN {X 0,Y 319.575,Z 239.676,A -85,B 0,C 180,E1 -15338.008,E2 -15338.008} C_VEL
LIN {X 0,Y 319.527,Z 239.682,A -85,B 0,C 180,E1 -15341.597,E2 -15341.597} C_VEL
LIN {X 0,Y 319.517,Z 239.686,A -85,B 0,C 180,E1 -15345.262,E2 -15345.262} C_VEL
LIN {X 0,Y 319.502,Z 239.692,A -85,B 0,C 180,E1 -15348.707,E2 -15348.707} C_VEL
LIN {X 0,Y 319.548,Z 239.686,A -85,B 0,C 180,E1 -15352.352,E2 -15352.352} C_VEL
LIN {X 0,Y 319.607,Z 239.826,A -85,B 0,C 180,E1 -15354.649,E2 -15354.649} C_VEL
LIN {X 0,Y 321.658,Z 248.473,A -85,B 0,C 180,E1 -15357.531,E2 -15357.531} C_VEL
LIN {X 0,Y 330.43,Z 268.498,A -85,B 0,C 180,E1 -15358.859,E2 -15358.859} C_VEL
LIN {X 0,Y 331.967,Z 272.99,A -85,B 0,C 180,E1 -15359.106,E2 -15359.106} C_VEL
LIN {X 0,Y 333.681,Z 280.643,A -85,B 0,C 180,E1 -15359.441,E2 -15359.441} C_VEL
LIN {X 0,Y 331.689,Z 356.191,A -85,B 0,C 180,E1 -15361.095,E2 -15361.095} C_VEL
LIN {X 0,Y 330.873,Z 370.176,A -85,B 0,C 180,E1 -15361.667,E2 -15361.667} C_VEL
LIN {X 0,Y 329.902,Z 382.124,A -85,B 0,C 180,E1 -15362.397,E2 -15362.397} C_VEL
LIN {X 0,Y 328.562,Z 393.365,A -85,B 0,C 180,E1 -15363.308,E2 -15363.308} C_VEL
LIN {X 0,Y 327.034,Z 405.026,A -85,B 0,C 180,E1 -15364.545,E2 -15364.545} C_VEL
LIN {X 0,Y 325.408,Z 415.489,A -85,B 0,C 180,E1 -15365.943,E2 -15365.943} C_VEL
LIN {X 0,Y 324,Z 424.014,A -85,B 0,C 180,E1 -15367.355,E2 -15367.355} C_VEL
LIN {X 0,Y 322.374,Z 433.209,A -85,B 0,C 180,E1 -15369.252,E2 -15369.252} C_VEL
LIN {X 0,Y 321.037,Z 440.586,A -85,B 0,C 180,E1 -15371.162,E2 -15371.162} C_VEL
LIN {X 0,Y 320.108,Z 445.566,A -85,B 0,C 180,E1 -15372.759,E2 -15372.759} C_VEL
LIN {X 0,Y 319.253,Z 450.381,A -85,B 0,C 180,E1 -15374.683,E2 -15374.683} C_VEL
LIN {X 0,Y 318.644,Z 454.06,A -85,B 0,C 180,E1 -15376.609,E2 -15376.609} C_VEL
LIN {X 0,Y 318.134,Z 456.707,A -85,B 0,C 180,E1 -15378.532,E2 -15378.532} C_VEL
LIN {X 0,Y 317.893,Z 457.948,A -85,B 0,C 180,E1 -15379.813,E2 -15379.813} C_VEL
LIN {X 0,Y 317.812,Z 458.779,A -85,B 0,C 180,E1 -15381.095,E2 -15381.095} C_VEL
LIN {X 0,Y 317.847,Z 459.184,A -85,B 0,C 180,E1 -15383.653,E2 -15383.653} C_VEL
LIN {X 0,Y 317.831,Z 458.054,A -85,B 0,C 180,E1 -15386.196,E2 -15386.196} C_VEL
LIN {X 0,Y 317.914,Z 455.263,A -85,B 0,C 180,E1 -15388.733,E2 -15388.733} C_VEL
LIN {X 0,Y 318.241,Z 452.06,A -85,B 0,C 180,E1 -15390.633,E2 -15390.633} C_VEL
LIN {X 0,Y 318.623,Z 447.809,A -85,B 0,C 180,E1 -15392.528,E2 -15392.528} C_VEL
LIN {X 0,Y 319.35,Z 441.38,A -85,B 0,C 180,E1 -15394.734,E2 -15394.734} C_VEL
LIN {X 0,Y 320.199,Z 434.329,A -85,B 0,C 180,E1 -15396.617,E2 -15396.617} C_VEL
LIN {X 0,Y 321.412,Z 425.539,A -85,B 0,C 180,E1 -15398.488,E2 -15398.488} C_VEL
LIN {X 0,Y 322.651,Z 415.55,A -85,B 0,C 180,E1 -15400.194,E2 -15400.194} C_VEL
LIN {X 0,Y 323.818,Z 405.33,A -85,B 0,C 180,E1 -15401.581,E2 -15401.581} C_VEL
LIN {X 0,Y 324.959,Z 394.004,A -85,B 0,C 180,E1 -15402.808,E2 -15402.808} C_VEL
LIN {X 0,Y 325.987,Z 382.167,A -85,B 0,C 180,E1 -15403.802,E2 -15403.802} C_VEL
LIN {X 0,Y 326.77,Z 369.47,A -85,B 0,C 180,E1 -15404.583,E2 -15404.583} C_VEL
LIN {X 0,Y 327.296,Z 356.303,A -85,B 0,C 180,E1 -15405.131,E2 -15405.131} C_VEL
LIN {X 0,Y 328.761,Z 293.661,A -85,B 0,C 180,E1 -15406.509,E2 -15406.509} C_VEL
LIN {X 0,Y 328.956,Z 276.933,A -85,B 0,C 180,E1 -15406.879,E2 -15406.879} C_VEL
LIN {X 0,Y 325.805,Z 260.334,A -85,B 0,C 180,E1 -15407.472,E2 -15407.472} C_VEL
LIN {X 0,Y 321.324,Z 247.976,A -85,B 0,C 180,E1 -15408.11,E2 -15408.11} C_VEL
LIN {X 0,Y 319.626,Z 239.673,A -85,B 0,C 180,E1 -15410.682,E2 -15410.682} C_VEL
LIN {X 0,Y 319.586,Z 239.678,A -85,B 0,C 180,E1 -15414.697,E2 -15414.697} C_VEL
LIN {X 0,Y 319.56,Z 239.68,A -85,B 0,C 180,E1 -15418.936,E2 -15418.936} C_VEL
LIN {X 0,Y 319.537,Z 239.681,A -85,B 0,C 180,E1 -15421.193,E2 -15421.193} C_VEL
LIN {X 0,Y 318.844,Z 239.769,A -85,B 0,C 180,E1 -15422.245,E2 -15422.245} C_VEL
LIN {X 0,Y 315.995,Z 240.121,A -85,B 0,C 180,E1 -15423.956,E2 -15423.956} C_VEL
LIN {X 0,Y 313.603,Z 240.419,A -85,B 0,C 180,E1 -15425.343,E2 -15425.343} C_VEL
LIN {X 0,Y 312.586,Z 240.548,A -85,B 0,C 180,E1 -15426.417,E2 -15426.417} C_VEL
LIN {X 0,Y 312.507,Z 240.552,A -85,B 0,C 180,E1 -15426.781,E2 -15426.781} C_VEL
LIN {X 0,Y 312.491,Z 240.562,A -85,B 0,C 180,E1 -15430.709,E2 -15430.709} C_VEL
LIN {X 0,Y 312.475,Z 240.56,A -85,B 0,C 180,E1 -15434.205,E2 -15434.205} C_VEL
LIN {X 0,Y 312.486,Z 240.558,A -85,B 0,C 180,E1 -15437.918,E2 -15437.918} C_VEL
LIN {X 0,Y 312.499,Z 240.558,A -85,B 0,C 180,E1 -15440.971,E2 -15440.971} C_VEL
LIN {X 0,Y 312.533,Z 240.553,A -85,B 0,C 180,E1 -15444.22,E2 -15444.22} C_VEL
LIN {X 0,Y 312.505,Z 240.549,A -85,B 0,C 180,E1 -15447.334,E2 -15447.334} C_VEL
LIN {X 0,Y 312.545,Z 240.55,A -85,B 0,C 180,E1 -15451.279,E2 -15451.279} C_VEL
LIN {X 0,Y 312.586,Z 240.546,A -85,B 0,C 180,E1 -15454.711,E2 -15454.711} C_VEL
LIN {X 0,Y 312.588,Z 240.536,A -85,B 0,C 180,E1 -15457.529,E2 -15457.529} C_VEL
LIN {X 0,Y 312.639,Z 240.537,A -85,B 0,C 180,E1 -15461.656,E2 -15461.656} C_VEL
LIN {X 0,Y 312.695,Z 240.529,A -85,B 0,C 180,E1 -15465.686,E2 -15465.686} C_VEL
LIN {X 0,Y 312.686,Z 240.524,A -85,B 0,C 180,E1 -15469.641,E2 -15469.641} C_VEL
LIN {X 0,Y 312.8,Z 240.517,A -85,B 0,C 180,E1 -15472.252,E2 -15472.252} C_VEL
LIN {X 0,Y 312.705,Z 240.533,A -85,B 0,C 180,E1 -15474.842,E2 -15474.842} C_VEL
LIN {X 0,Y 312.935,Z 240.499,A -85,B 0,C 180,E1 -15477.425,E2 -15477.425} C_VEL
LIN {X 0,Y 313.083,Z 240.483,A -85,B 0,C 180,E1 -15480,E2 -15480} C_VEL
LIN {X 0,Y 312.933,Z 240.506,A -85,B 0,C 180,E1 -15482.574,E2 -15482.574} C_VEL
LIN {X 0,Y 312.911,Z 240.508,A -85,B 0,C 180,E1 -15486.448,E2 -15486.448} C_VEL
LIN {X 0,Y 312.788,Z 240.52,A -85,B 0,C 180,E1 -15489.049,E2 -15489.049} C_VEL
LIN {X 0,Y 312.635,Z 240.54,A -85,B 0,C 180,E1 -15492.991,E2 -15492.991} C_VEL
LIN {X 0,Y 312.622,Z 240.54,A -85,B 0,C 180,E1 -15495.651,E2 -15495.651} C_VEL
LIN {X 0,Y 312.539,Z 240.549,A -85,B 0,C 180,E1 -15499.713,E2 -15499.713} C_VEL
LIN {X 0,Y 312.524,Z 240.555,A -85,B 0,C 180,E1 -15502.78,E2 -15502.78} C_VEL
LIN {X 0,Y 312.533,Z 240.55,A -85,B 0,C 180,E1 -15505.909,E2 -15505.909} C_VEL
LIN {X 0,Y 312.5,Z 240.555,A -85,B 0,C 180,E1 -15509.655,E2 -15509.655} C_VEL
LIN {X 0,Y 312.519,Z 240.553,A -85,B 0,C 180,E1 -15513.689,E2 -15513.689} C_VEL
LIN {X 0,Y 312.514,Z 240.554,A -85,B 0,C 180,E1 -15517.387,E2 -15517.387} C_VEL
LIN {X 0,Y 312.44,Z 240.567,A -85,B 0,C 180,E1 -15520.717,E2 -15520.717} C_VEL
LIN {X 0,Y 312.451,Z 240.565,A -85,B 0,C 180,E1 -15524.21,E2 -15524.21} C_VEL
LIN {X 0,Y 312.483,Z 240.557,A -85,B 0,C 180,E1 -15527.919,E2 -15527.919} C_VEL
LIN {X 0,Y 312.506,Z 240.556,A -85,B 0,C 180,E1 -15531.917,E2 -15531.917} C_VEL
LIN {X 0,Y 312.533,Z 240.555,A -85,B 0,C 180,E1 -15534.221,E2 -15534.221} C_VEL
LIN {X 0,Y 312.504,Z 240.558,A -85,B 0,C 180,E1 -15537.334,E2 -15537.334} C_VEL
LIN {X 0,Y 312.522,Z 240.705,A -85,B 0,C 180,E1 -15538.782,E2 -15538.782} C_VEL
LIN {X 0,Y 314.893,Z 251.534,A -85,B 0,C 180,E1 -15542.051,E2 -15542.051} C_VEL
LIN {X 0,Y 316.405,Z 260.71,A -85,B 0,C 180,E1 -15544.686,E2 -15544.686} C_VEL
LIN {X 0,Y 316.036,Z 264.022,A -85,B 0,C 180,E1 -15545.56,E2 -15545.56} C_VEL
LIN {X 0,Y 320.737,Z 294.68,A -85,B 0,C 180,E1 -15546.631,E2 -15546.631} C_VEL
LIN {X 0,Y 321.918,Z 304.515,A -85,B 0,C 180,E1 -15546.941,E2 -15546.941} C_VEL
LIN {X 0,Y 320.442,Z 373.215,A -85,B 0,C 180,E1 -15548.489,E2 -15548.489} C_VEL
LIN {X 0,Y 319.651,Z 387.01,A -85,B 0,C 180,E1 -15549.067,E2 -15549.067} C_VEL
LIN {X 0,Y 318.65,Z 399.38,A -85,B 0,C 180,E1 -15549.842,E2 -15549.842} C_VEL
LIN {X 0,Y 317.361,Z 412.047,A -85,B 0,C 180,E1 -15550.935,E2 -15550.935} C_VEL
LIN {X 0,Y 316.028,Z 423.324,A -85,B 0,C 180,E1 -15552.195,E2 -15552.195} C_VEL
LIN {X 0,Y 314.812,Z 433.601,A -85,B 0,C 180,E1 -15553.652,E2 -15553.652} C_VEL
LIN {X 0,Y 313.873,Z 441.806,A -85,B 0,C 180,E1 -15555.078,E2 -15555.078} C_VEL
LIN {X 0,Y 312.701,Z 450.862,A -85,B 0,C 180,E1 -15557.012,E2 -15557.012} C_VEL
LIN {X 0,Y 311.852,Z 458.153,A -85,B 0,C 180,E1 -15558.956,E2 -15558.956} C_VEL
LIN {X 0,Y 311.268,Z 463.977,A -85,B 0,C 180,E1 -15560.906,E2 -15560.906} C_VEL
LIN {X 0,Y 310.917,Z 468.553,A -85,B 0,C 180,E1 -15562.858,E2 -15562.858} C_VEL
LIN {X 0,Y 310.724,Z 472.025,A -85,B 0,C 180,E1 -15564.809,E2 -15564.809} C_VEL
LIN {X 0,Y 310.72,Z 473.757,A -85,B 0,C 180,E1 -15566.109,E2 -15566.109} C_VEL
LIN {X 0,Y 310.683,Z 475.074,A -85,B 0,C 180,E1 -15567.407,E2 -15567.407} C_VEL
LIN {X 0,Y 310.658,Z 475.994,A -85,B 0,C 180,E1 -15568.704,E2 -15568.704} C_VEL
LIN {X 0,Y 310.691,Z 476.513,A -85,B 0,C 180,E1 -15570,E2 -15570} C_VEL
LIN {X 0,Y 310.677,Z 476.295,A -85,B 0,C 180,E1 -15572.593,E2 -15572.593} C_VEL
LIN {X 0,Y 310.699,Z 475.609,A -85,B 0,C 180,E1 -15573.891,E2 -15573.891} C_VEL
LIN {X 0,Y 310.775,Z 473.95,A -85,B 0,C 180,E1 -15575.71,E2 -15575.71} C_VEL
LIN {X 0,Y 311.208,Z 469.935,A -85,B 0,C 180,E1 -15578.441,E2 -15578.441} C_VEL
LIN {X 0,Y 311.837,Z 465.827,A -85,B 0,C 180,E1 -15580.387,E2 -15580.387} C_VEL
LIN {X 0,Y 312.85,Z 459.555,A -85,B 0,C 180,E1 -15582.652,E2 -15582.652} C_VEL
LIN {X 0,Y 314.214,Z 452.743,A -85,B 0,C 180,E1 -15584.574,E2 -15584.574} C_VEL
LIN {X 0,Y 315.729,Z 444.273,A -85,B 0,C 180,E1 -15586.488,E2 -15586.488} C_VEL
LIN {X 0,Y 317.192,Z 435.578,A -85,B 0,C 180,E1 -15588.071,E2 -15588.071} C_VEL
LIN {X 0,Y 319.056,Z 424.89,A -85,B 0,C 180,E1 -15589.628,E2 -15589.628} C_VEL
LIN {X 0,Y 320.709,Z 414.259,A -85,B 0,C 180,E1 -15590.861,E2 -15590.861} C_VEL
LIN {X 0,Y 322.35,Z 402.361,A -85,B 0,C 180,E1 -15591.923,E2 -15591.923} C_VEL
LIN {X 0,Y 323.666,Z 389.998,A -85,B 0,C 180,E1 -15592.754,E2 -15592.754} C_VEL
LIN {X 0,Y 324.682,Z 377.253,A -85,B 0,C 180,E1 -15593.353,E2 -15593.353} C_VEL
LIN {X 0,Y 325.295,Z 363.789,A -85,B 0,C 180,E1 -15593.728,E2 -15593.728} C_VEL
LIN {X 0,Y 326.653,Z 305.108,A -85,B 0,C 180,E1 -15595.027,E2 -15595.027} C_VEL
LIN {X 0,Y 322.049,Z 279.442,A -85,B 0,C 180,E1 -15596.085,E2 -15596.085} C_VEL
LIN {X 0,Y 319.412,Z 268.119,A -85,B 0,C 180,E1 -15596.625,E2 -15596.625} C_VEL
LIN {X 0,Y 317.667,Z 263.602,A -85,B 0,C 180,E1 -15596.949,E2 -15596.949} C_VEL
LIN {X 0,Y 315.849,Z 254.372,A -85,B 0,C 180,E1 -15599.797,E2 -15599.797} C_VEL
LIN {X 0,Y 313.311,Z 243.813,A -85,B 0,C 180,E1 -15603.259,E2 -15603.259} C_VEL
LIN {X 0,Y 312.523,Z 240.554,A -85,B 0,C 180,E1 -15604.403,E2 -15604.403} C_VEL
LIN {X 0,Y 312.494,Z 240.56,A -85,B 0,C 180,E1 -15608.08,E2 -15608.08} C_VEL
LIN {X 0,Y 312.491,Z 240.56,A -85,B 0,C 180,E1 -15610.709,E2 -15610.709} C_VEL
LIN {X 0,Y 312.452,Z 240.564,A -85,B 0,C 180,E1 -15614.21,E2 -15614.21} C_VEL
LIN {X 0,Y 312.456,Z 240.565,A -85,B 0,C 180,E1 -15617.924,E2 -15617.924} C_VEL
LIN {X 0,Y 312.484,Z 240.558,A -85,B 0,C 180,E1 -15621.922,E2 -15621.922} C_VEL
LIN {X 0,Y 312.531,Z 240.553,A -85,B 0,C 180,E1 -15624.22,E2 -15624.22} C_VEL
LIN {X 0,Y 312.502,Z 240.552,A -85,B 0,C 180,E1 -15627.334,E2 -15627.334} C_VEL
LIN {X 0,Y 312.525,Z 240.549,A -85,B 0,C 180,E1 -15631.286,E2 -15631.286} C_VEL
LIN {X 0,Y 312.555,Z 240.542,A -85,B 0,C 180,E1 -15634.708,E2 -15634.708} C_VEL
LIN {X 0,Y 312.565,Z 240.548,A -85,B 0,C 180,E1 -15637.527,E2 -15637.527} C_VEL
LIN {X 0,Y 312.583,Z 240.547,A -85,B 0,C 180,E1 -15641.653,E2 -15641.653} C_VEL
LIN {X 0,Y 312.687,Z 240.536,A -85,B 0,C 180,E1 -15645.686,E2 -15645.686} C_VEL
LIN {X 0,Y 312.702,Z 240.532,A -85,B 0,C 180,E1 -15649.642,E2 -15649.642} C_VEL
LIN {X 0,Y 312.868,Z 240.504,A -85,B 0,C 180,E1 -15652.254,E2 -15652.254} C_VEL
LIN {X 0,Y 312.709,Z 240.529,A -85,B 0,C 180,E1 -15654.842,E2 -15654.842} C_VEL
LIN {X 0,Y 312.986,Z 240.488,A -85,B 0,C 180,E1 -15658.713,E2 -15658.713} C_VEL
LIN {X 0,Y 312.987,Z 240.498,A -85,B 0,C 180,E1 -15661.287,E2 -15661.287} C_VEL
LIN {X 0,Y 312.703,Z 240.532,A -85,B 0,C 180,E1 -15665.158,E2 -15665.158} C_VEL
LIN {X 0,Y 312.803,Z 240.511,A -85,B 0,C 180,E1 -15667.748,E2 -15667.748} C_VEL
LIN {X 0,Y 312.665,Z 240.536,A -85,B 0,C 180,E1 -15671.672,E2 -15671.672} C_VEL
LIN {X 0,Y 312.668,Z 240.533,A -85,B 0,C 180,E1 -15674.865,E2 -15674.865} C_VEL
LIN {X 0,Y 312.611,Z 240.538,A -85,B 0,C 180,E1 -15679.226,E2 -15679.226} C_VEL
LIN {X 0,Y 312.547,Z 240.542,A -85,B 0,C 180,E1 -15682.789,E2 -15682.789} C_VEL
LIN {X 0,Y 312.598,Z 240.538,A -85,B 0,C 180,E1 -15685.933,E2 -15685.933} C_VEL
LIN {X 0,Y 312.54,Z 240.549,A -85,B 0,C 180,E1 -15689.651,E2 -15689.651} C_VEL
LIN {X 0,Y 312.521,Z 240.553,A -85,B 0,C 180,E1 -15693.689,E2 -15693.689} C_VEL
LIN {X 0,Y 312.539,Z 240.554,A -85,B 0,C 180,E1 -15697.384,E2 -15697.384} C_VEL
LIN {X 0,Y 312.491,Z 240.56,A -85,B 0,C 180,E1 -15700.709,E2 -15700.709} C_VEL
LIN {X 0,Y 312.474,Z 240.563,A -85,B 0,C 180,E1 -15704.206,E2 -15704.206} C_VEL
LIN {X 0,Y 312.46,Z 240.565,A -85,B 0,C 180,E1 -15707.924,E2 -15707.924} C_VEL
LIN {X 0,Y 312.486,Z 240.567,A -85,B 0,C 180,E1 -15711.922,E2 -15711.922} C_VEL
LIN {X 0,Y 312.536,Z 240.696,A -85,B 0,C 180,E1 -15714.051,E2 -15714.051} C_VEL
LIN {X 0,Y 314.54,Z 248.866,A -85,B 0,C 180,E1 -15716.815,E2 -15716.815} C_VEL
LIN {X 0,Y 323.653,Z 269.191,A -85,B 0,C 180,E1 -15718.241,E2 -15718.241} C_VEL
LIN {X 0,Y 325.921,Z 275.371,A -85,B 0,C 180,E1 -15718.608,E2 -15718.608} C_VEL
LIN {X 0,Y 327.398,Z 282.434,A -85,B 0,C 180,E1 -15718.918,E2 -15718.918} C_VEL
LIN {X 0,Y 325.305,Z 356.399,A -85,B 0,C 180,E1 -15720.561,E2 -15720.561} C_VEL
LIN {X 0,Y 324.46,Z 370.379,A -85,B 0,C 180,E1 -15721.143,E2 -15721.143} C_VEL
LIN {X 0,Y 323.442,Z 382.323,A -85,B 0,C 180,E1 -15721.885,E2 -15721.885} C_VEL
LIN {X 0,Y 321.959,Z 394.363,A -85,B 0,C 180,E1 -15722.891,E2 -15722.891} C_VEL
LIN {X 0,Y 320.325,Z 405.981,A -85,B 0,C 180,E1 -15724.162,E2 -15724.162} C_VEL
LIN {X 0,Y 318.67,Z 416.207,A -85,B 0,C 180,E1 -15725.574,E2 -15725.574} C_VEL
LIN {X 0,Y 317.038,Z 425.454,A -85,B 0,C 180,E1 -15727.174,E2 -15727.174} C_VEL
LIN {X 0,Y 315.39,Z 434.426,A -85,B 0,C 180,E1 -15729.112,E2 -15729.112} C_VEL
LIN {X 0,Y 314.022,Z 441.612,A -85,B 0,C 180,E1 -15731.064,E2 -15731.064} C_VEL
LIN {X 0,Y 312.88,Z 447.307,A -85,B 0,C 180,E1 -15733.022,E2 -15733.022} C_VEL
LIN {X 0,Y 312.067,Z 451.773,A -85,B 0,C 180,E1 -15734.99,E2 -15734.99} C_VEL
LIN {X 0,Y 311.426,Z 455.146,A -85,B 0,C 180,E1 -15736.958,E2 -15736.958} C_VEL
LIN {X 0,Y 311.091,Z 456.813,A -85,B 0,C 180,E1 -15738.269,E2 -15738.269} C_VEL
LIN {X 0,Y 310.743,Z 458.937,A -85,B 0,C 180,E1 -15740.891,E2 -15740.891} C_VEL
LIN {X 0,Y 310.708,Z 459.361,A -85,B 0,C 180,E1 -15742.2,E2 -15742.2} C_VEL
LIN {X 0,Y 310.725,Z 459.202,A -85,B 0,C 180,E1 -15744.384,E2 -15744.384} C_VEL
LIN {X 0,Y 310.738,Z 458.311,A -85,B 0,C 180,E1 -15746.109,E2 -15746.109} C_VEL
LIN {X 0,Y 310.741,Z 457.146,A -85,B 0,C 180,E1 -15747.407,E2 -15747.407} C_VEL
LIN {X 0,Y 311.037,Z 453.587,A -85,B 0,C 180,E1 -15750,E2 -15750} C_VEL
LIN {X 0,Y 311.386,Z 449.741,A -85,B 0,C 180,E1 -15751.94,E2 -15751.94} C_VEL
LIN {X 0,Y 311.965,Z 444.775,A -85,B 0,C 180,E1 -15753.875,E2 -15753.875} C_VEL
LIN {X 0,Y 312.684,Z 438.546,A -85,B 0,C 180,E1 -15755.805,E2 -15755.805} C_VEL
LIN {X 0,Y 313.786,Z 430.739,A -85,B 0,C 180,E1 -15757.723,E2 -15757.723} C_VEL
LIN {X 0,Y 314.905,Z 422.785,A -85,B 0,C 180,E1 -15759.312,E2 -15759.312} C_VEL
LIN {X 0,Y 316.068,Z 413.1,A -85,B 0,C 180,E1 -15760.895,E2 -15760.895} C_VEL
LIN {X 0,Y 317.373,Z 402.306,A -85,B 0,C 180,E1 -15762.306,E2 -15762.306} C_VEL
LIN {X 0,Y 318.405,Z 391.763,A -85,B 0,C 180,E1 -15763.401,E2 -15763.401} C_VEL
LIN {X 0,Y 319.498,Z 378.916,A -85,B 0,C 180,E1 -15764.421,E2 -15764.421} C_VEL
LIN {X 0,Y 320.266,Z 365.993,A -85,B 0,C 180,E1 -15765.163,E2 -15765.163} C_VEL
LIN {X 0,Y 320.692,Z 353.972,A -85,B 0,C 180,E1 -15765.613,E2 -15765.613} C_VEL
LIN {X 0,Y 322.327,Z 278.063,A -85,B 0,C 180,E1 -15767.297,E2 -15767.297} C_VEL
LIN {X 0,Y 319.354,Z 262.413,A -85,B 0,C 180,E1 -15767.873,E2 -15767.873} C_VEL
